	//Alarm
	TON_ComAlarm(IN:= MesWarningCom  , PT:= ParamTempoComAlarm, Q=>MesDataExd.MesAlarmCom) ;	// Alarms if ALL TRAM MODBUS did not work and timeout of 15s

// ALARM CODE //
	FB_AlarmCodeManager(
		bAlarm1			:= InvAlarm[1],		// All module are in alarm Inverter 1
		bAlarm2			:= InvAlarm[2],		// All module are in alarm Inverter 2
		bAlarm3			:= InvAlarm[3],		// All module are in alarm Inverter 3
		bAlarm4			:= MesDataExd.MesAlarmCom, 	//AT Least one Com error with 18 x Modules during more than 30s         
		bAlarm5			:= FALSE,
		bAlarm6			:= FALSE,
		bAlarm7			:= FALSE,
		bAlarm8			:= FALSE,
		bAlarm9			:= FALSE,
		bAlarm10		:= FALSE,
		bAlarm11		:= FALSE, 
		bAlarm12		:= FALSE, 
		bAlarm13		:= FALSE, 
		bAlarm14		:= FALSE, 													// 
		bAlarm15		:= FALSE,
		wAlarmCode		=> MesDataExd.MesAlarmCode);

// WARNING CODE //
	FB_AlarmCodeManager(
 		bAlarm1			:= INVWarning[1],//AT LEast one moduls of inverter 1 in alarm
		bAlarm2			:= INVWarning[2],//AT LEast one moduls of inverter 2 in alarm
		bAlarm3			:= INVWarning[3],//AT LEast one moduls of inverter 3 in alarm
		bAlarm4			:= MesWarningCom,//AT Least one Com error with 18 x Modules
		bAlarm5			:= FALSE, 		
		bAlarm6			:= FALSE, 		
		bAlarm7			:= FALSE, 
		bAlarm8			:= FALSE, 
		bAlarm9			:= FALSE, 
		bAlarm10		:= FALSE, 
		bAlarm11		:= FALSE, 
		bAlarm12		:= FALSE, 
		bAlarm13		:= FALSE, 
		bAlarm14		:= FALSE, 
		bAlarm15		:= FALSE, 
		wAlarmCode		=> MesDataExd.MesWarningCode);	

		
// EVENT CODE //
	FB_AlarmCodeManager(
		bAlarm1			:= RS_StartStop.Q1, 			// Start command
		bAlarm2			:= NOT RS_StartStop.Q1, 		// Stop command
		bAlarm3			:= FALSE,	
		bAlarm4			:= FALSE, 	
		bAlarm5			:= FALSE, 
		bAlarm6			:= FALSE, 
		bAlarm7			:= FALSE, 
		bAlarm8			:= FALSE, 
		bAlarm9			:= FALSE, 
		bAlarm10		:= FALSE, 
		bAlarm11		:= FALSE, 
		bAlarm12		:= FALSE, 
		bAlarm13		:= FALSE, 
		bAlarm14		:= FALSE, 
		bAlarm15		:= FALSE, 
		wAlarmCode		=> MesDataExd.MesEventCode);
END_METHOD

METHOD M_CP
//////////////////
//  Emulator
/////////////////

VAR 
	// Method local variables (reinitialized at each cycle) 
	
END_VAR


SUPER^.M_CP() ; 




Trig_Cmd_Read(CLK:=IN_CmdToggleRead);
//Trig_Cmd_Write(CLK:=IN_CmdToggleWrite);
//	
IF Trig_Cmd_Read.Q THEN
	IN_CmdToggleRead := FALSE;
	MesDataExd.AX_INV[1].MesData.MesCP_Read := NOT MesDataExd.AX_INV[1].MesData.MesCP_Read;
END_IF
//
//
//IF Trig_Cmd_Write.Q THEN
//	IN_CmdToggleWrite := FALSE;
//	MesDataExd.MesData.MesCP_Write := NOT MesDataExd.MesData.MesCP_Write;
//END_IF
END_METHOD

{attribute 'object_name' := 'M_Curtail'}
METHOD M_Curtail
//////////////////
// Write Curtail Command through modbus to PV inverters.  
//////////////////
VAR 
	// Method local variables (reinitialized at each cycle) 
	Threshold 			 : INT:=5 ;					// (0-100) Change percentage of Range to trigger the write command. 

	CHECK				 : BOOL; 					// Check if changes. 
	WriteCmdInvMode		: BOOL;

	MesSEPAM	: ProtectRelay_S48;
	

END_VAR




MesDataExd.OUT_SetptTanPhi := IN_SetptTanPhi ; 
MesDataExd.OUT_SetptP		:= ParamPn ; 
MesDataExd.OUT_CmdStart	:= TRUE ;
MesDataExd.OUT_CmdStop	:= FALSE ;

	
OUT_CmdSetpt420_IO := 32767- REAL_TO_INT((32767 * (MesDataExd.OUT_SetptTanPhi+0.484)/(0.968))  );		// ? ? 
 
SUPER^.M_Curtail() ;
END_METHOD

METHOD M_Execute
//////////////////
//  Method Calls 
/////////////////

VAR 
	// Method local variables (reinitialized at each cycle) 

END_VAR
IF  bInit THEN
	M_Init();
END_IF

(*
TP_Read(In := NOT(TP_Read.Q) AND NOT ReadBusy);
RTrig(CLK := TP_Read.Q);
ClockRead := RTrig.Q;
*)
SUPER^.M_Execute() ;
END_METHOD

METHOD M_Init
VAR_INPUT
END_VAR

VAR

END_VAR
//ParamPn := 990 ;
bInit := FALSE;
//FB_ModbusRTU() ;
AX_bRead[1] := TRUE ; 
(*
FB_ModbusRead(
	Inquantity		:= Nb_DataBlockModules,
	InUnitID 		:= ParamUnitID ,
	InTimeout		:= ParamTimeout,
	InInterfaceSub	:= FALSE,
	InFunctionRead	:= TRUE	);
	
	*)
END_METHOD

{attribute 'object_name' := 'M_Read'}
METHOD M_Read
//////////
// Read Method for SMA : Modbus reading
//////////
VAR
	// Method local variables (reinitialized at each cycle) 
	MW_32MLE		: FB_WordsToFloat32MLE;
	AX_bRead_init 		: ARRAY[0..18] OF BOOL; 
	KK					: BYTE;						 // Index to loop over modbus blocks. 	
	JJ					: BYTE;

	InclockRead: INT;
END_VAR


IF MesDataExd.AX_INV[1].MesData.MesCP_Read  THEN	







OutFBCompleteted:=FALSE;

// MODBUS REQUEST//


	
		// Reset Structure output. 
		//InputStructRead	:= InputStructRead_Null; 
		//
		//InputStructRead.InFunction := ParamFunctionReadModbus;
		//InputStructRead.InQuantity := Nb_DataBlockModules;	
		//
		//InputStructRead.OutBusy := ADR(ReadBusy);
		//InputStructRead.OutError := ADR(ReadError);
		//InputStructRead.OutCompleted := ADR(bReadCompleted);

		FB_ModbusRTU.ReadRTU1(
				InClockRead := NOT ClockRead AND AX_bRead[Steps],
				InStartAddr :=  AX_Start_Adresse[Steps],
				InQuantity := Nb_DataBlockModules,
				InUnitID := ParamUnitID,
				InTimeout := T#1500MS,
				InAddrDest := ADR(MesBlock_Temp[Steps]),
				InFunctionRead := ParamFunctionReadModbus,
				InInterfaceSub	:= FALSE 
			);
		
		IF  FB_ModbusRTU.ReadRTU1.OutBusy AND AX_bRead[Steps]THEN 
			AX_bRead[Steps] 	:= FALSE; 
		
		END_IF	
	
		RTrigI(CLK:= FB_ModbusRTU.ReadRTU1.TmpError );
		IF FB_ModbusRTU.ReadRTU1.OutbCompleted THEN

			Steps:= SEL(Steps >= 18 , Steps +1 , 1) ;
			AX_bRead[Steps] 	:= TRUE;
			ReadError := FALSE ; 
			
		ELSIF NOT FB_ModbusRTU.ReadRTU1.OutBusy  AND  RTrigI.Q THEN
			Steps:= SEL(Steps >= 18 , Steps +1 , 1) ;
			AX_bRead[Steps] 	:= TRUE;
			ReadError := TRUE ; 
		
		END_IF

//FB_ModbusRTU() ; 

	CalAllCompleted := AX_bRead[1] AND AX_bRead[2] AND AX_bRead[3] AND AX_bRead[4] AND AX_bRead[5] AND AX_bRead[6]; 
	CalAllCompleted := CalAllCompleted AND AX_bRead[7] AND AX_bRead[8] AND AX_bRead[9] AND AX_bRead[10] AND AX_bRead[11] AND AX_bRead[12];
	CalAllCompleted := CalAllCompleted AND AX_bRead[13] AND AX_bRead[14] AND AX_bRead[15] AND AX_bRead[16] AND AX_bRead[17] AND AX_bRead[18];	
	
	CalAllBugged	:= AX_bRead[1] OR AX_bRead[2] OR AX_bRead[3] OR AX_bRead[4] OR AX_bRead[5] OR AX_bRead[6];
	CalAllBugged 	:= CalAllBugged OR AX_bRead[7] OR AX_bRead[8] OR AX_bRead[9] OR AX_bRead[10] OR AX_bRead[11] OR AX_bRead[12];
	CalAllBugged 	:= CalAllBugged OR AX_bRead[13] OR AX_bRead[14] OR AX_bRead[15] OR AX_bRead[16] OR AX_bRead[17] OR AX_bRead[18];	
	
	
	OutFBCompleteted := CalAllCompleted	;
	TON_AllBugged(IN := NOT CalAllBugged, pt := T#10S);
	TRIG_AllBugged(CLK := TON_AllBugged.Q);
	IF TRIG_AllBugged.Q THEN
		TON_AllBugged(IN := FALSE);
		AX_bRead[Steps] := TRUE;
	END_IF

	////CHECK IF ALL MODBUS REQUESTS ARE FINISHED
	IF (CalAllCompleted) THEN
		////RESETING CLOCK READ FOR EACH REQUEST
		//AX_bRead:= AX_bRead_init;
		CalAllCompleted := FALSE;
	END_IF
	MesTempPos[1] := 0;
	MesTempPos[2] := 0;
	// PROPERTIES UPDATE
	// MODBUS BLOCKS SEPARATION	& PROPERTIES UPDATE
		//INVERTER 01 - Module
	
	
	JJ := 1 ; 
	
	FOR KK := 1 TO 18 BY 1 DO
		
		IF KK =1 THEN
			//InverterNumber := 1 ;
			InverterNumber := 1;// on constate un décalage de deux bloque avec cette méthode. Ainsi , l'adresse correspondant à INV1 (AX_Start_Adresse[1] , donne un résultat dans le block 3 Block_Temp[3]. 

		END_IF

		DecalageInvModule := SEL(((KK+0) MOD 6) =0 , (KK+0) MOD 6  , 6);//KK - (6*(InverterNumber-1)) ;
			
		//Word on 1 register To INT 
		MesDataExd.AX_INV[InverterNumber].AX_PowerCol[DecalageInvModule].MesSN 				:= WORD_TO_INT(MesBlock_Temp[KK][0]);
		MesDataExd.AX_INV[InverterNumber].AX_PowerCol[DecalageInvModule].MesID_Type 	:= WORD_TO_INT(MesBlock_Temp[KK][1]);
		MesDataExd.AX_INV[InverterNumber].AX_PowerCol[DecalageInvModule].MesID_StateGlobal		:= WORD_TO_INT(MesBlock_Temp[KK][2]);
		MesDataExd.AX_INV[InverterNumber].AX_PowerCol[DecalageInvModule].MesIDState	    := WORD_TO_INT(MesBlock_Temp[KK][3]);
		MesDataExd.AX_INV[InverterNumber].AX_PowerCol[DecalageInvModule].MesAlarmID		:= WORD_TO_INT(MesBlock_Temp[KK][4]);
		// 5 et 6 is blanck
		//Word on 2 register To Float 32
		//Module Information
			//Part1
		MW_32MLE(InFirstWord:=MesBlock_Temp[KK][7],InSecondWord:=MesBlock_Temp[KK][8],OutCalReal	=>MesDataExd.AX_INV[InverterNumber].AX_PowerCol[DecalageInvModule].MesEDay);
		MW_32MLE(InFirstWord:=MesBlock_Temp[KK][9],InSecondWord:=MesBlock_Temp[KK][10],OutCalReal	=>MesDataExd.AX_INV[InverterNumber].AX_PowerCol[DecalageInvModule].MesETot);
		MW_32MLE(InFirstWord:=MesBlock_Temp[KK][11],InSecondWord:=MesBlock_Temp[KK][12],OutCalReal  =>MesDataExd.AX_INV[InverterNumber].AX_PowerCol[DecalageInvModule].MesEPartial);
		MW_32MLE(InFirstWord:=MesBlock_Temp[KK][13],InSecondWord:=MesBlock_Temp[KK][14],OutCalReal  =>MesDataExd.AX_INV[InverterNumber].AX_PowerCol[DecalageInvModule].MesEWeek);
		MW_32MLE(InFirstWord:=MesBlock_Temp[KK][15],InSecondWord:=MesBlock_Temp[KK][16],OutCalReal  =>MesDataExd.AX_INV[InverterNumber].AX_PowerCol[DecalageInvModule].MesEMonth);
		MW_32MLE(InFirstWord:=MesBlock_Temp[KK][17],InSecondWord:=MesBlock_Temp[KK][18],OutCalReal  =>MesDataExd.AX_INV[InverterNumber].AX_PowerCol[DecalageInvModule].MesEYear);
			//Part2                                                                                                      
		MW_32MLE(InFirstWord:=MesBlock_Temp[KK][33],InSecondWord:=MesBlock_Temp[KK][34],OutCalReal  =>MesDataExd.AX_INV[InverterNumber].AX_PowerCol[DecalageInvModule].MesTemp_Inv);
		MW_32MLE(InFirstWord:=MesBlock_Temp[KK][35],InSecondWord:=MesBlock_Temp[KK][36],OutCalReal  =>MesDataExd.AX_INV[InverterNumber].AX_PowerCol[DecalageInvModule].MesTemp_Supply);
		MW_32MLE(InFirstWord:=MesBlock_Temp[KK][37],InSecondWord:=MesBlock_Temp[KK][38],OutCalReal  =>MesDataExd.AX_INV[InverterNumber].AX_PowerCol[DecalageInvModule].MesTemp_Headsink);
		MW_32MLE(InFirstWord:=MesBlock_Temp[KK][39],InSecondWord:=MesBlock_Temp[KK][40],OutCalReal  =>MesDataExd.AX_INV[InverterNumber].AX_PowerCol[DecalageInvModule].MesTemp_T2);
		MW_32MLE(InFirstWord:=MesBlock_Temp[KK][41],InSecondWord:=MesBlock_Temp[KK][42],OutCalReal  =>MesDataExd.AX_INV[InverterNumber].AX_PowerCol[DecalageInvModule].MesTemp_T3);
		

		// Detect Communication Error : MesID_StateGlobal = 0 , MesAlarmID = 0 , Temp_Inv = 0 
		IF MesDataExd.AX_INV[InverterNumber].AX_PowerCol[DecalageInvModule].MesTemp_Inv = 0 
			AND MesDataExd.AX_INV[InverterNumber].AX_PowerCol[DecalageInvModule].MesID_StateGlobal = 0 
			AND MesDataExd.AX_INV[InverterNumber].AX_PowerCol[DecalageInvModule].MesAlarmID = 0 THEN  
				MesDataExd.AX_INV[InverterNumber].AX_PowerCol[DecalageInvModule].MesAlarmID := 8 ; 
		END_IF
		
	
		IF  MesDataExd.AX_INV[InverterNumber].AX_PowerCol[DecalageInvModule].MesID_Type = 1  THEN
			//Slave
			MW_32MLE(InFirstWord:=MesBlock_Temp[KK][19],InSecondWord:=MesBlock_Temp[KK][20],OutCalReal=>MesDataExd.AX_INV[InverterNumber].AX_PowerCol[DecalageInvModule].MesV);
			MW_32MLE(InFirstWord:=MesBlock_Temp[KK][21],InSecondWord:=MesBlock_Temp[KK][22],OutCalReal=>MesTempPSlave[JJ][4]);
			MesDataExd.AX_INV[InverterNumber].AX_PowerCol[DecalageInvModule].MesI := MesTempPSlave[JJ][4] ; 
			MW_32MLE(InFirstWord:=MesBlock_Temp[KK][23],InSecondWord:=MesBlock_Temp[KK][24],OutCalReal=>MesTempPSlave[JJ][1]);
			MesDataExd.AX_INV[InverterNumber].AX_PowerCol[DecalageInvModule].MesData.MesP := MesTempPSlave[JJ][1];
			MW_32MLE(InFirstWord:=MesBlock_Temp[KK][25],InSecondWord:=MesBlock_Temp[KK][26],OutCalReal=>MesDataExd.AX_INV[InverterNumber].AX_PowerCol[DecalageInvModule].MesData.MesFreq);
			MW_32MLE(InFirstWord:=MesBlock_Temp[KK][27],InSecondWord:=MesBlock_Temp[KK][28],OutCalReal=>MesTempPSlave[JJ][2]);
			MesDataExd.AX_INV[InverterNumber].AX_PowerCol[DecalageInvModule].MesData.MesPdc := MesTempPSlave[JJ][2];
			MW_32MLE(InFirstWord:=MesBlock_Temp[KK][29],InSecondWord:=MesBlock_Temp[KK][30],OutCalReal=>MesDataExd.AX_INV[InverterNumber].AX_PowerCol[DecalageInvModule].MesData.MesUdc);
			MW_32MLE(InFirstWord:=MesBlock_Temp[KK][31],InSecondWord:=MesBlock_Temp[KK][32],OutCalReal=>MesTempPSlave[JJ][3]);
			MesDataExd.AX_INV[InverterNumber].AX_PowerCol[DecalageInvModule].MesData.MesIdc := MesTempPSlave[JJ][3] ;
		ELSE      
			//Master                                                                                                               
			MW_32MLE(InFirstWord:=MesBlock_Temp[KK][55],InSecondWord:=MesBlock_Temp[KK][56],OutCalReal=>MesDataExd.AX_INV[InverterNumber].AX_PowerCol[DecalageInvModule].MesV);
			MW_32MLE(InFirstWord:=MesBlock_Temp[KK][57],InSecondWord:=MesBlock_Temp[KK][58],OutCalReal=>MesTempPMaster[JJ][4]);
			MW_32MLE(InFirstWord:=MesBlock_Temp[KK][59],InSecondWord:=MesBlock_Temp[KK][60],OutCalReal=>MesTempPMaster[JJ][1]);
			//MesDataExd.AX_INV[InverterNumber].AX_PowerCol[DecalageInvModule].MesP := MesTempPMaster[JJ][1];
			MW_32MLE(InFirstWord:=MesBlock_Temp[KK][25],InSecondWord:=MesBlock_Temp[KK][26],OutCalReal=>MesDataExd.AX_INV[InverterNumber].AX_PowerCol[DecalageInvModule].MesData.MesFreq);
			MW_32MLE(InFirstWord:=MesBlock_Temp[KK][61],InSecondWord:=MesBlock_Temp[KK][62],OutCalReal=>MesTempPMaster[JJ][2]);
			//MesDataExd.AX_INV[InverterNumber].AX_PowerCol[DecalageInvModule].MesPdc := MesTempPMaster[JJ][2];
			MW_32MLE(InFirstWord:=MesBlock_Temp[KK][63],InSecondWord:=MesBlock_Temp[KK][64],OutCalReal=>MesDataExd.AX_INV[InverterNumber].AX_PowerCol[DecalageInvModule].MesData.MesUdc);
			MW_32MLE(InFirstWord:=MesBlock_Temp[KK][65],InSecondWord:=MesBlock_Temp[KK][66],OutCalReal=>MesTempPMaster[JJ][3]); 
			MesTempPos[JJ] := DecalageInvModule ; 	// Relative Number of master module 
		END_IF
		
		IF KK MOD 2 =0 THEN
			IF Master_slave_Calculation AND MesTempPos[JJ]>0 THEN
				MesDataExd.AX_INV[InverterNumber].AX_PowerCol[MesTempPos[JJ]].MesData.MesP := MesTempPMaster[JJ][1]- MesTempPSlave[JJ][1];	// P
				MesDataExd.AX_INV[InverterNumber].AX_PowerCol[MesTempPos[JJ]].MesData.MesPdc := MesTempPMaster[JJ][2]- MesTempPSlave[JJ][2];	// Pdc
				MesDataExd.AX_INV[InverterNumber].AX_PowerCol[MesTempPos[JJ]].MesData.MesIdc :=MesTempPMaster[JJ][3]- MesTempPSlave[JJ][3];	// Idc
				MesDataExd.AX_INV[InverterNumber].AX_PowerCol[MesTempPos[JJ]].MesI := MesTempPMaster[JJ][4]- MesTempPSlave[JJ][4];	// I

				IF MesDataExd.AX_INV[InverterNumber].AX_PowerCol[MesTempPos[JJ]].MesData.MesP < 0 THEN 
					MesDataExd.AX_INV[InverterNumber].AX_PowerCol[MesTempPos[JJ]].MesData.MesP := 0 ; 
					MesDataExd.AX_INV[InverterNumber].AX_PowerCol[MesTempPos[JJ]].MesData.MesPdc := 0 ; 
					MesDataExd.AX_INV[InverterNumber].AX_PowerCol[MesTempPos[JJ]].MesData.MesIdc := 0 ; 
					MesDataExd.AX_INV[InverterNumber].AX_PowerCol[MesTempPos[JJ]].MesI := 0 ;
					MesDataExd.AX_INV[InverterNumber].AX_PowerCol[MesTempPos[JJ]].MesAlarmID := 8  ;  // Com error with master
					
				ELSIF MesDataExd.AX_INV[InverterNumber].AX_PowerCol[MesTempPos[JJ]].MesData.MesP > 50 THEN // Higher than Pnom 
					MesDataExd.AX_INV[InverterNumber].AX_PowerCol[MesTempPos[JJ]].MesAlarmID := 88  ; // Com error with Slave device 
				END_IF
				
			ELSIF MesTempPos[JJ]>0 THEN 
				MesDataExd.AX_INV[InverterNumber].AX_PowerCol[MesTempPos[JJ]].MesData.MesP := MesTempPMaster[JJ][1];	// P
				MesDataExd.AX_INV[InverterNumber].AX_PowerCol[MesTempPos[JJ]].MesData.MesPdc := MesTempPMaster[JJ][2];	// Pdc
				MesDataExd.AX_INV[InverterNumber].AX_PowerCol[MesTempPos[JJ]].MesData.MesIdc := MesTempPMaster[JJ][3];	// Idc				
				MesDataExd.AX_INV[InverterNumber].AX_PowerCol[MesTempPos[JJ]].MesI := MesTempPMaster[JJ][4];	// I					
				
			END_IF
			JJ := JJ +1;		
		END_IF
		
		// RACK informations
		IF DecalageInvModule = 6  THEN
			
			MW_32MLE(InFirstWord:=MesBlock_Temp[KK][43],InSecondWord:=MesBlock_Temp[KK][44],OutCalReal=>MesDataExd.AX_INV[InverterNumber].MesEDay);
			MW_32MLE(InFirstWord:=MesBlock_Temp[KK][45],InSecondWord:=MesBlock_Temp[KK][46],OutCalReal=>MesDataExd.AX_INV[InverterNumber].MesETot);
			MW_32MLE(InFirstWord:=MesBlock_Temp[KK][47],InSecondWord:=MesBlock_Temp[KK][48],OutCalReal=>MesDataExd.AX_INV[InverterNumber].MesEPartial);
			MW_32MLE(InFirstWord:=MesBlock_Temp[KK][49],InSecondWord:=MesBlock_Temp[KK][50],OutCalReal=>MesDataExd.AX_INV[InverterNumber].MesEWeek);
			MW_32MLE(InFirstWord:=MesBlock_Temp[KK][51],InSecondWord:=MesBlock_Temp[KK][52],OutCalReal=>MesDataExd.AX_INV[InverterNumber].MesEMonth);
			MW_32MLE(InFirstWord:=MesBlock_Temp[KK][53],InSecondWord:=MesBlock_Temp[KK][54],OutCalReal=>MesDataExd.AX_INV[InverterNumber].MesEYear);
			InverterNumber := SEL(InverterNumber=3 , InverterNumber + 1,1);
		END_IF
		
	END_FOR;
	
	//Calculation of Master/slave power
(*
	IF FALSE AND Master_slave_Calculation THEN
		//Inverter 1
			//P
			MesDataExd.AX_INV[1].AX_PowerCol[MesTempPos[1]].MesP := MesTempPMaster[1][1]- MesTempPSlave[1][1];
			MesDataExd.AX_INV[1].AX_PowerCol[MesTempPos[2]].MesP := MesTempPMaster[2][1]- MesTempPSlave[2][1];
			MesDataExd.AX_INV[1].AX_PowerCol[MesTempPos[3]].MesP := MesTempPMaster[3][1]- MesTempPSlave[3][1];
			//Pdc
			MesDataExd.AX_INV[1].AX_PowerCol[MesTempPos[1]].MesPdc := MesTempPMaster[1][2]- MesTempPSlave[1][2];
			MesDataExd.AX_INV[1].AX_PowerCol[MesTempPos[2]].MesPdc := MesTempPMaster[2][2]- MesTempPSlave[2][2];
			MesDataExd.AX_INV[1].AX_PowerCol[MesTempPos[3]].MesPdc := MesTempPMaster[3][2]- MesTempPSlave[3][2];
			
		//Inverter 2
			//P
			MesDataExd.AX_INV[2].AX_PowerCol[MesTempPos[4]].MesP := MesTempPMaster[4][1]- MesTempPSlave[4][1];
			MesDataExd.AX_INV[2].AX_PowerCol[MesTempPos[5]].MesP := MesTempPMaster[5][1]- MesTempPSlave[5][1];
			MesDataExd.AX_INV[2].AX_PowerCol[MesTempPos[6]].MesP := MesTempPMaster[6][1]- MesTempPSlave[6][1];
			//Pdc    
			MesDataExd.AX_INV[2].AX_PowerCol[MesTempPos[4]].MesPdc := MesTempPMaster[4][2]- MesTempPSlave[4][2];
			MesDataExd.AX_INV[2].AX_PowerCol[MesTempPos[5]].MesPdc := MesTempPMaster[5][2]- MesTempPSlave[5][2];
			MesDataExd.AX_INV[2].AX_PowerCol[MesTempPos[6]].MesPdc := MesTempPMaster[6][2]- MesTempPSlave[6][2];
		             
		//Inverter 3  
			//P       
			MesDataExd.AX_INV[3].AX_PowerCol[MesTempPos[7]].MesP := MesTempPMaster[7][1]- MesTempPSlave[7][1];
			MesDataExd.AX_INV[3].AX_PowerCol[MesTempPos[8]].MesP := MesTempPMaster[8][1]- MesTempPSlave[8][1];
			MesDataExd.AX_INV[3].AX_PowerCol[MesTempPos[9]].MesP := MesTempPMaster[9][1]- MesTempPSlave[9][1];
			//Pdc     
			MesDataExd.AX_INV[3].AX_PowerCol[MesTempPos[7]].MesPdc := MesTempPMaster[7][2]- MesTempPSlave[7][2];
			MesDataExd.AX_INV[3].AX_PowerCol[MesTempPos[8]].MesPdc := MesTempPMaster[8][2]- MesTempPSlave[8][2];
			MesDataExd.AX_INV[3].AX_PowerCol[MesTempPos[9]].MesPdc := MesTempPMaster[9][2]- MesTempPSlave[9][2];
	ELSE
		//Inverter 1
			MesDataExd.AX_INV[1].AX_PowerCol[MesTempPos[1]].MesP := MesTempPMaster[1][1];
			MesDataExd.AX_INV[1].AX_PowerCol[MesTempPos[2]].MesP := MesTempPMaster[2][1];
			MesDataExd.AX_INV[1].AX_PowerCol[MesTempPos[3]].MesP := MesTempPMaster[3][1];
			//Pdc     
			MesDataExd.AX_INV[1].AX_PowerCol[MesTempPos[1]].MesPdc := MesTempPMaster[1][2];
			MesDataExd.AX_INV[1].AX_PowerCol[MesTempPos[2]].MesPdc := MesTempPMaster[2][2];
			MesDataExd.AX_INV[1].AX_PowerCol[MesTempPos[3]].MesPdc := MesTempPMaster[3][2];
		//Inverter 2  
			//P      
			MesDataExd.AX_INV[2].AX_PowerCol[MesTempPos[4]].MesP := MesTempPMaster[4][1];
			MesDataExd.AX_INV[2].AX_PowerCol[MesTempPos[5]].MesP := MesTempPMaster[5][1];
			MesDataExd.AX_INV[2].AX_PowerCol[MesTempPos[6]].MesP := MesTempPMaster[6][1];
			//Pdc     
			MesDataExd.AX_INV[2].AX_PowerCol[MesTempPos[4]].MesPdc := MesTempPMaster[4][2];
			MesDataExd.AX_INV[2].AX_PowerCol[MesTempPos[5]].MesPdc := MesTempPMaster[5][2];
			MesDataExd.AX_INV[2].AX_PowerCol[MesTempPos[6]].MesPdc := MesTempPMaster[6][2];
		             
		//Inverter 3  
			//P      
			MesDataExd.AX_INV[3].AX_PowerCol[MesTempPos[7]].MesP := MesTempPMaster[7][1];
			MesDataExd.AX_INV[3].AX_PowerCol[MesTempPos[8]].MesP := MesTempPMaster[8][1];
			MesDataExd.AX_INV[3].AX_PowerCol[MesTempPos[9]].MesP := MesTempPMaster[9][1];
			//Pdc     
			MesDataExd.AX_INV[3].AX_PowerCol[MesTempPos[7]].MesPdc := MesTempPMaster[7][2];
			MesDataExd.AX_INV[3].AX_PowerCol[MesTempPos[8]].MesPdc := MesTempPMaster[8][2];
			MesDataExd.AX_INV[3].AX_PowerCol[MesTempPos[9]].MesPdc := MesTempPMaster[9][2];
	END_IF	
	*)
//Addition des puissance
	FOR KK:= 1 TO 3 DO 
		MesDataExd.AX_INV[KK].MesData.MesP := 0 ; 
		MesDataExd.AX_INV[KK].MesData.MesI := 0 ; 
		MesDataExd.AX_INV[KK].MesData.MesPdc := 0 ; 
		MesDataExd.AX_INV[KK].MesData.MesFreq :=  0 ; 
		MesDataExd.AX_INV[KK].MesData.MesIdc := 0  ; 
		MesDataExd.AX_INV[KK].MesData.MesV := 0  ; 		
		MesDataExd.AX_INV[KK].MesData.MesUdc := 0  ; 		
 		MesDataExd.AX_INV[KK].MesData.MesTemp	:= 0 ; 
		MesDataExd.AX_INV[KK].MesData.ParamPn := ParamPn/3 ; 
		
		FOR InclockRead:= 1 TO 6 DO 
			MesDataExd.AX_INV[KK].MesData.MesP  	:= MesDataExd.AX_INV[KK].MesData.MesP +	MesDataExd.AX_INV[KK].AX_PowerCol[InclockRead].MesData.MesP ;					
			MesDataExd.AX_INV[KK].MesData.MesPdc  	:= MesDataExd.AX_INV[KK].MesData.MesPdc +	MesDataExd.AX_INV[KK].AX_PowerCol[InclockRead].MesData.MesPdc ;					
			MesDataExd.AX_INV[KK].MesData.MesI  	:= MesDataExd.AX_INV[KK].MesData.MesI +	MesDataExd.AX_INV[KK].AX_PowerCol[InclockRead].MesI ;					
			MesDataExd.AX_INV[KK].MesData.MesFreq 	:= MAX(MesDataExd.AX_INV[KK].MesData.MesFreq , MesDataExd.AX_INV[KK].AX_PowerCol[InclockRead].MesData.MesFreq) ; 
			MesDataExd.AX_INV[KK].MesData.MesIdc  	:= MesDataExd.AX_INV[KK].MesData.MesIdc +	MesDataExd.AX_INV[KK].AX_PowerCol[InclockRead].MesData.MesIdc ;			
			MesDataExd.AX_INV[KK].MesData.MesUdc 	:= MAX(MesDataExd.AX_INV[KK].MesData.MesUdc , MesDataExd.AX_INV[KK].AX_PowerCol[InclockRead].MesData.MesUdc) ; 		
			MesDataExd.AX_INV[KK].MesData.MesV 	:= MAX(MesDataExd.AX_INV[KK].MesData.MesV , MesDataExd.AX_INV[KK].AX_PowerCol[InclockRead].MesV) ; 
			MesDataExd.AX_INV[KK].MesData.MesTemp 	:= MAX(MesDataExd.AX_INV[KK].MesData.MesTemp , MesDataExd.AX_INV[KK].AX_PowerCol[InclockRead].MesTemp_Inv) ; 	
		END_FOR
	

	END_FOR

END_IF
END_METHOD

METHOD M_StateManager
//////////////////
// Detect which is the state of the inverter. IF loss of communication MesState =0 , the last inverter state is kept .  
/////////////////

VAR 
	// Method local variables (reinitialized at each cycle) 

	
	KK: INT;
	LL: INT;

	MesAll_Start	: BOOL;
	MesALO_Fault 	: BOOL;
	MesALO_Stopped	: BOOL;
	MesAll_Fault: BOOL;
	
	
	CalIDState_PowerCol: INT;
	CalNbPowerCol: INT;	
	
	
END_VAR
MesDataExd.MesNbInvConnected := 0  ; 
FOR KK:= 1  TO 3 DO 
	MesDataExd.AX_INV[KK].MesNbPowerColConnected := 0  ; 
	FOR LL:=1 TO 6 DO 
		
		CalIDState_PowerCol := MesDataExd.AX_INV[KK].AX_PowerCol[LL].MesID_StateGlobal ; 
	
		IF CalIDState_PowerCol = 6 THEN 
			MesDataExd.AX_INV[KK].MesNbPowerColConnected  := MesDataExd.AX_INV[KK].MesNbPowerColConnected + 1 ; 
		END_IF

	END_FOR	
	
	IF MesDataExd.AX_INV[KK].MesNbPowerColConnected> 0  THEN 
		MesDataExd.MesNbInvConnected := MesDataExd.MesNbInvConnected  + 1 ;  
	END_IF

END_FOR

// Check over all the powercolonnes 
//O=Stopped, 1 = MPPT, 2 = Sleeping, 3 = Starting, 4 = Throttled, 5 = Shutting down, 6 = Fault, 7 = Standby

FOR KK := 1 TO CstNbInv_PTR_G DO
	MesAll_Start := TRUE;
	MesAll_Fault := TRUE ;
	FOR LL := 1 TO CstNbPowerCol_INV_G DO 
		MesAll_Start := MesAll_Start AND MesDataExd.AX_INV[KK].AX_PowerCol[LL].MesIDState = 45;
		MesALO_Fault := MesALO_Fault OR MesDataExd.AX_INV[KK].AX_PowerCol[LL].MesAlarmID > 0;
		MesAll_Fault := MesAll_Fault AND MesDataExd.AX_INV[KK].AX_PowerCol[LL].MesAlarmID > 0;
		MesALO_Stopped := MesALO_Stopped OR 
			(MesDataExd.AX_INV[KK].AX_PowerCol[LL].MesIDState = 45 AND MesDataExd.AX_INV[KK].AX_PowerCol[LL].MesAlarmID > 0);
	END_FOR
	
	MesDataExd.AX_INV[KK].MesData.MesState := 0;
	
	IF MesDataExd.AX_INV[KK].MesNbPowerColConnected > 0 THEN 
		IF MesDataExd.AX_INV[KK].MesData.MesP > 0.01 THEN 
			MesDataExd.AX_INV[KK].MesData.MesState.1 := TRUE ; // MPPT 
		ELSE 
			MesDataExd.AX_INV[KK].MesData.MesState.7 := TRUE ;  // Standby 
		END_IF 	
	ELSE 
		IF MesAll_Fault THEN 
			MesDataExd.AX_INV[KK].MesData.MesState.6 := TRUE ; // Fault 
		ELSE 
			MesDataExd.AX_INV[KK].MesData.MesState.0 := TRUE ; // Off 
		END_IF
	END_IF

END_FOR

MesDataExd.MesState 			:= 0  ; // At Cluster level
IF MesDataExd.MesNbInvConnected=0   THEN  // 
	// OFF State  
	MesDataExd.MesState.0 		:= 1 ; 
	
ELSE
	// ON State
	MesDataExd.MesState.2 		:= 1 ;
	
END_IF



SUPER^.M_StateManager() ;
END_METHOD

END_FUNCTION_BLOCK

// ---- 00_FunctionsBlocks/Beckhoff/Communication/ModbusRTU/FB_ModbusRTU.TcPOU
FUNCTION_BLOCK FB_ModbusRTU
// Send Modbus Read Request for the first element of the buffer . Then remove the first line when executed ( busy)  and move all the other line to the left. Position 2 becomes position 1 , ...
VAR CONSTANT
	NbElementsBuffer				: UINT := 20;
	
END_VAR
VAR_INPUT PERSISTENT
	ParamTimeout					: TIME := T#500MS;
	ParamInterfaceSub				: BOOL;
END_VAR
VAR
	Buffer 							: ARRAY[1..NbElementsBuffer] OF Struct_InputRTU ; // Buffer to store actions
	Priority 						: ARRAY[1..NbElementsBuffer] OF UINT; // Array to store priorities
	InitialStruct 					: Struct_InputRTU;
	bInit 							: BOOL;
	ReadRTU1						: FB_ReadModbusRTU_V2;

	KK : UINT;
	
	pBoolNull						: BOOL;
	pIntNull						: INT;
	pArrayNull						: BYTE;

	R_TRIG_Error					: R_TRIG ;
	F_Trig_busy						: F_TRIG;
END_VAR

IF NOT bInit THEN
	// Empty all structures . 
	M_Init();
ELSE
	
		// ATTENTION , IL NE FAUT PAS ENVOYER UN NOUVEAU MODBUS TANT QUE LE PRECEDENT N EST PAS FINI DE TRAITER .DE MEME IL NE FAUT PAS QUE LE CYCLE D AJOUT DU FIFO SOIT PLUS RAPIDE QUE LE TRAITEMENT DU RTU 
		// TEmpo de 30 s apres une alarmes avant de refaire un essai . il ne faudrait pas que ca bloque les autres commandes .  

		IF priority[1] <> 0 THEN

			ReadRTU1(
				InClockRead := TRUE,
				InStartAddr := Buffer[1].InStartAddr,
				InQuantity := Buffer[1].InQuantity,
				InUnitID := Buffer[1].InUnitID,
				InTimeout := ParamTimeout,
				InAddrDest := Buffer[1].InBuffer,
				InFunctionRead := Buffer[1].InFunction,
				InInterfaceSub	:= ParamInterfaceSub 
			);
		END_IF
		
		
		
		MEMCPY(destAddr := Buffer[1].OutBusy, srcAddr := ADR(ReadRTU1.OutBusy), n := SIZEOF(ReadRTU1.OutBusy));		

		//R_TRIG_Error(CLK:= ReadRTU1.OutErrorMbRead) ; 
		F_Trig_busy(clk := ReadRTU1.OutBusy);
		IF F_Trig_busy.Q THEN	// La lecture s 'est terminée par une erreur ou correcteemnt, on passe à l'element du buffer suivant . 
			MEMCPY(destAddr := Buffer[1].OutError, srcAddr := ADR(ReadRTU1.OutErrorMbRead), n := SIZEOF(ReadRTU1.OutErrorMbRead)); // Copy the errOR  
			MEMCPY(destAddr := Buffer[1].OutErrorId, srcAddr := ADR(ReadRTU1.OutErrorId), n := SIZEOF(ReadRTU1.OutErrorId));
			MEMCPY(destAddr := Buffer[1].OutCompleted, srcAddr := ADR(ReadRTU1.OutbCompleted), n := SIZEOF(ReadRTU1.OutbCompleted));	
			ReadRTU1.InClockRead := FALSE ; 
			ReadRTU1.Reset		:= TRUE ; 
			M_DeleteAction(InLigne := 1);
			//R_TRIG_Error(CLK:= FALSE ) ; 
			
		END_IF
END_IF

METHOD M_AddAction_FIFO : UINT //Method to add an element with a priority using FIFO strategy

VAR_INPUT
	InStruct 		: Struct_InputRTU;		// Structure input
	InPriority 		: UINT;					// Strategy input
END_VAR
VAR_OUTPUT
	OutBusy 		: BOOL;					// Output state of the Method
	OutError 		: BOOL;					// Output error of the Method
	OutErrorID 		: UINT;					//1: Empty input 2: Full Buffer
	OutCompleted 	: BOOL;					// Output state of the Method : not busy and no error
END_VAR
VAR
	KK 				: UINT;
	LineToDelete	: UINT;
END_VAR
OutError 	:= FALSE;
OutBusy 	:= TRUE;

IF NOT (CheckStruct(InStruct1 := InitialStruct, InStruct2 := InStruct)) AND InPriority <> 0 THEN 			// Check that we don't input an empty value
	IF CheckStruct(InStruct1 := buffer[NbElementsBuffer], InStruct2 := InitialStruct) THEN 			// Check that the buffer isn't already full
		FOR KK := 1 TO NbElementsBuffer - 1 DO
			IF NOT CheckStruct(InStruct1 := buffer[NbElementsBuffer-KK], InStruct2 := InitialStruct) AND Priority[NbElementsBuffer-KK] > InPriority THEN 			// If the next position isn't empty  
				buffer[NbElementsBuffer-KK+1] := buffer[NbElementsBuffer-KK]; 		// I replace this position by the next  ( CE PREMIER IF N EST PAS EXECUTER SI TOUTES LES PRIORITES SONT IDENTIQUES . )
				Priority[NbElementsBuffer -KK +1 ] := Priority[NbElementsBuffer-KK];
			ELSE
				IF NOT CheckStruct(InStruct1 := buffer[NbElementsBuffer-KK], InStruct2 := InitialStruct) THEN		// Detect for buffer element that is not empty and assign new element to read to it. 
					buffer[NbElementsBuffer-KK+1] 	:= InStruct;
					M_AddAction_FIFO 				:= NbElementsBuffer-KK+1;
					Priority[NbElementsBuffer-KK+1] := InPriority;
					OutCompleted 		:= TRUE;
					EXIT ;
				END_IF
			END_IF
		END_FOR
		IF NOT Outcompleted THEN
			buffer[1] := InStruct;
			Priority[1] := InPriority;
			OutCompleted := TRUE;
			M_AddAction_Fifo := 1;
		END_IF
	ELSE
		OutErrorID 	:= 2;
		OutError 	:= TRUE;
	END_IF
ELSE
	OutErrorID 	:= 1;
	OutError 	:= TRUE;
END_IF
IF M_VerifActions(OutLigne=>LineToDelete) THEN	// Verifie si il  n ya pas deux fois la meme ligne , sinon, supprime les lignes en doubles . En pratique, forcement la derniere ligne . 
	M_DeleteAction(InLigne := LineToDelete);
END_IF
OutBusy := FALSE;
END_METHOD

METHOD M_DeleteAction : BOOL
VAR_INPUT
	InLigne 	: UINT;			// Input Ligne to delete
END_VAR
VAR_OUTPUT
	OutBusy 		: BOOL;					// Output state of the Method
	OutError 		: BOOL;					// Output error of the Method
	OutErrorID 		: UINT;					// 1: InLigne greater than Buffer size, 2: The buffer ligne is already empty, 3: The buffer is full
	OutCompleted 	: BOOL;					// Output state of the Method : not busy and no error
	
END_VAR

VAR
	KK 				: UINT;
END_VAR
IF InLigne <= NbElementsBuffer THEN // Check the InLigne is in the range of the buffer
	IF NOT checkstruct(InStruct1 := buffer[InLigne], InStruct2 := InitialStruct) THEN	// Check that the buffer ligne is not already empty
		IF checkstruct(InStruct1 := buffer[NbElementsBuffer], InStruct2 := InitialStruct)THEN //check that the buffer is not full
			FOR KK := InLigne TO NbElementsBuffer -1 DO
				Buffer[KK] := buffer[KK + 1] ;
				Priority[KK] := Priority[KK + 1] ;
			END_FOR
		ELSE
			OutError := TRUE;
			OutBusy := FALSE;
			OutCompleted := FALSE;
			OutErrorID := 3;
		END_IF
	ELSE
		OutError := TRUE;
		OutCompleted := FALSE;
		OutBusy := TRUE;
		OutErrorID := 2;
		
	END_IF
ELSE
	OutCompleted := FALSE;
	OutError := TRUE;
	OutBusy := FALSE;
	OutErrorID := 1;
END_IF
END_METHOD

METHOD M_Init : BOOL
VAR
	InStruct : Struct_InputRTU;
END_VAR

// Initialize the structure with empty elements. 

InitialStruct.InBuffer := ADR(pArrayNull);
InitialStruct.OutBusy := ADR(pBoolNull);
InitialStruct.OutCompleted := ADR(pBoolNull);
InitialStruct.OutError := ADR(pBoolNull);
InitialStruct.OutErrorId := ADR(pIntNull);
FOR KK := 1 TO NbElementsBuffer DO 
	Buffer[KK] := InitialStruct;
END_FOR	

bInit := TRUE;
END_METHOD

METHOD M_VerifActions : BOOL // Verifies there is not repeat in the liste : TRUE = At least 2 elements are the same
VAR_OUTPUT
	OutLigne 	 : UINT;
END_VAR

VAR
	KK: UINT;
	JJ: UINT;
	CheckStructValue : BOOL;
END_VAR
FOR KK := 1 TO NbElementsBuffer DO
	FOR JJ := 1 + KK TO NbElementsBuffer DO
		IF CheckStruct(InStruct1 := InitialStruct, instruct2 := buffer[KK]) THEN
			EXIT;
		ELSE
			CheckStructValue :=  checkstruct(InStruct1 := buffer[JJ], InStruct2 := buffer[KK]);
			M_VerifActions := M_VerifActions OR (CheckStructValue ) ;
			OutLigne := SEL(CheckStructValue AND Priority[KK]> priority[JJ], KK, JJ);
		END_IF
	END_FOR
END_FOR
END_METHOD

END_FUNCTION_BLOCK

// ---- 00_FunctionsBlocks/Beckhoff/Communication/ModbusRTU/FB_ReadModbusRTU_V2.TcPOU
FUNCTION_BLOCK FB_ReadModbusRTU_V2
/////////////////////////////////////////////////////////////////////// 
///////Read Modbus RTU on Rising Edge of Trigger ClockRead ////////
//If there is lost of communication, ParamNbAlms then if still 
//error wait ParamTimeRetry then loop 
//Version : V1.1
///////////////////////////////////////////////////////////////////////

VAR_INPUT
	InClockRead 			: BOOL;  		// Boolean to start the read
	InStartAddr				: WORD;  		// First address of the block
	InQuantity			    : WORD;	 		// Quantity of registers to read
	InUnitID				: BYTE ; 		// Unit Id of the Slave to be read
	InTimeout 				: TIME:=T#2S;   // Timeout param for the read
	InAddrDest		        : POINTER TO BYTE;
	InInterfaceSub			: BOOL:=FALSE;   // Serial interface RS422/RS485 TYPE (0:EL6021,1:SUB9)
	InFunctionRead          : UINT;          // 0 := ReadInputRegs, 1 := ReadRegs 
	ParamEnableRetryPause	: BOOL ; 
	Reset					: BOOL ;
END_VAR

VAR_OUTPUT
	OutErrorMbRead  		: BOOL; 	                // Alarm if three modbus attempts failed.
	OutBusy					: BOOL;					    //Busy
	OutErrorId				: INT;            //Id number of the error based on TC
	OutbCompleted			: BOOL;
	TmpError				: BOOL;	
END_VAR

VAR
	//Parameters
	ParamNbAlms				: UINT := 3;				// Parameter for the number of retries before the alarme
	ParamTimeRetry 			: TIME:=T#30S;				//Time to wait before a retry
	
	//Instantiation of FB
	MB 						: ModbusRtuMaster_PcCOM; 		// Multiple registers reading FROM SUB9 Interface
	MB_EL					: ModbusRtuMasterV2_KL6x22B;  // Multiple registers reading FROM EL6021 Interface
	R_TRIG          		: R_TRIG; 					// Rising edge detection for the trigger.
	TempoRetry      		: TP;
	
	//Variables of the code 
	Step            		: INT; 		    			// Grafcet step
	AlarmCounter    		: UINT; 					// Alarm Counter. Incremennted if modbus errOR  Alarm if counter =3 , resetable.  
	bRetry          		: BOOL:= FALSE; 			// Boolean to denote the retries
	
	TmpBusy					: BOOL;
	TmpErrorId				: INT;	
	
	TON_ReadRTU						: TON; 
END_VAR

OutbCompleted:= FALSE;
// RESET //
	IF Reset THEN 
			AlarmCounter		:= MAX(0,AlarmCounter-1) ;	// on enleve 1 au compteur pour supprimer l'alamrme. 
			OutErrorId 			:= 0 ; 
			OutErrorMbRead 	:=FALSE;
			Reset 				:= FALSE;
	END_IF
	
// ALARM MANAGEMENT //
TempoRetry(PT := ParamTimeRetry);
IF AlarmCounter = ParamNbAlms THEN 
	OutErrorMbRead 	:=TRUE;
	bRetry := SEL(ParamEnableRetryPause , FALSE ,  TRUE);		// False = disable retry 	
ELSE
	bRetry := FALSE;
	
END_IF

	// MODBUS SEQUENCE //
	
	IF InInterfaceSub THEN 

		CASE step OF
			0://Idle
				R_TRIG(CLK := InClockRead);
				IF R_TRIG.Q THEN 
					R_TRIG(CLK := FALSE);
					Step :=1;
					OutBusy         := TRUE;
				END_IF
			1 ://Processing Reply  
				TON_ReadRTU(IN:= TRUE , PT:= InTimeout + T#100MS ) ; // Overlay timeout . 
				CASE InFunctionRead OF
					1: 
						MB.ReadCoils
						(
							UnitID := InUnitId, 
							Quantity := InQuantity, 
							MBAddr := InStartAddr, 
							cbLength := 2* InQuantity, 
							pMemoryAddr := InAddrDest, 
							Execute := TRUE, 
							Timeout := InTimeout,
							Error => TmpError,
							Busy => TmpBusy,
							ErrorId => TmpErrorId,
						);	
					2:
						MB.ReadInputStatus
						(
							UnitID := InUnitId, 
							Quantity := InQuantity, 
							MBAddr := InStartAddr, 
							cbLength := 2* InQuantity, 
							pMemoryAddr := InAddrDest, 
							Execute := TRUE, 
							Timeout := InTimeout,
							Error => TmpError,
							Busy => TmpBusy,
							ErrorId => TmpErrorId,
						);	
					3:
						MB.ReadRegs
						(
							UnitID := InUnitId, 
							Quantity := InQuantity, 
							MBAddr := InStartAddr, 
							cbLength := 2* InQuantity, 
							pMemoryAddr := InAddrDest, 
							Execute := TRUE, 
							Timeout := InTimeout,
							Error => TmpError,
							Busy => TmpBusy,
							ErrorId => TmpErrorId,
						  );
					4:
						MB.ReadInputRegs
						(
							UnitID := InUnitId, 
							Quantity := InQuantity, 
							MBAddr := InStartAddr, 
							cbLength := 2* InQuantity, 
							pMemoryAddr := InAddrDest, 
							Execute := TRUE, 
							Timeout := InTimeout,
							Error => TmpError,
							Busy => TmpBusy,
							ErrorId => TmpErrorId,
						);
					5:
						MB.WriteSingleCoil
						(
							UnitID := InUnitId, 
							Quantity := InQuantity, 
							MBAddr := InStartAddr, 
							cbLength := 2* InQuantity, 
							pMemoryAddr := InAddrDest, 
							Execute := TRUE, 
							Timeout := InTimeout,
							Error => TmpError,
							Busy => TmpBusy,
							ErrorId => TmpErrorId,
						);
					6:
						MB.WriteSingleRegister
						(
							UnitID := InUnitId, 
							Quantity := InQuantity, 
							MBAddr := InStartAddr, 
							cbLength := 2* InQuantity, 
							pMemoryAddr := InAddrDest, 
							Execute := TRUE, 
							Timeout := InTimeout,
							Error => TmpError,
							Busy => TmpBusy,
							ErrorId => TmpErrorId,
						);
					15:
						MB.WriteMultipleCoils
						(
							UnitID := InUnitId, 
							Quantity := InQuantity, 
							MBAddr := InStartAddr, 
							cbLength := 2* InQuantity, 
							pMemoryAddr := InAddrDest, 
							Execute := TRUE, 
							Timeout := InTimeout,
							Error => TmpError,
							Busy => TmpBusy,
							ErrorId => TmpErrorId,
						);
					16:
						MB.WriteRegs
						(
							UnitID := InUnitId, 
							Quantity := InQuantity, 
							MBAddr := InStartAddr, 
							cbLength := 2* InQuantity, 
							pMemoryAddr := InAddrDest, 
							Execute := TRUE, 
							Timeout := InTimeout,
							Error => TmpError,
							Busy => TmpBusy,
							ErrorId => TmpErrorId,
						);
				END_CASE
				
				IF NOT (TmpBusy) AND NOT (TmpError) THEN
					TempoRetry(In:= FALSE);
					TON_ReadRTU(IN:= FALSE ) ; 
					MB.ReadInputRegs(Execute:= FALSE);
					MB.ReadRegs(Execute:= FALSE);
					MB.ReadCoils(Execute:= FALSE);
					MB.ReadInputStatus(Execute:= FALSE);
					MB.WriteSingleCoil(Execute:= FALSE);
					MB.WriteSingleRegister(Execute:= FALSE);
					MB.WriteMultipleCoils(Execute:= FALSE);
					MB.WriteRegs(Execute:= FALSE);
					OutErrorId 		:= 0;
					OutErrorMbRead	:= FALSE;
					AlarmCounter	:= 0; // Reset counter after successful modbus read. 
					OutbCompleted 	:= TRUE ; 
					Step 			:= 0;
					OutBusy         := FALSE;
				ELSIF ((NOT (TmpBusy) AND TmpError) OR TON_ReadRTU.Q)  AND NOT(bRetry) THEN
	
					TempoRetry(In:= FALSE);
					bRetry := FALSE;
					MB.ReadCoils(Execute:= FALSE);
					MB.ReadInputRegs(Execute:= FALSE);
					MB.ReadInputStatus(Execute:= FALSE);
					MB.ReadRegs(Execute:= FALSE);
					MB.WriteSingleCoil(Execute:= FALSE);
					MB.WriteSingleRegister(Execute:= FALSE);
					MB.WriteMultipleCoils(Execute:= FALSE);
					MB.WriteRegs(Execute:= FALSE);
					AlarmCounter 	:= MIN(AlarmCounter + 1,3) ; 
					OutErrorId		:= SEL(TON_ReadRTU.Q , TmpErrorId ,250 );
					Step 			:= 0;
					TON_ReadRTU(IN:= FALSE ) ; 
					OutBusy         := FALSE;
				ELSIF NOT (TmpBusy) AND TmpError AND bRetry THEN
					MB.ReadInputRegs(Execute:= FALSE);
					MB.ReadRegs(Execute:= FALSE);
					MB.ReadCoils(Execute:= FALSE);
					MB.ReadInputStatus(Execute:= FALSE);
					MB.WriteSingleCoil(Execute:= FALSE);
					MB.WriteSingleRegister(Execute:= FALSE);
					MB.WriteMultipleCoils(Execute:= FALSE);
					MB.WriteRegs(Execute:= FALSE);
					step := 2;
					OutBusy         := FALSE;
				END_IF	
			2: 
				TempoRetry(In:= TRUE);		// LEAVE SOME TIME BEFORE NEW ATTEMPT . 
				IF NOT(TempoRetry.Q) THEN
					TempoRetry(In:= FALSE);
					//AlarmCounter := 0;
					step := 0;
					
				END_IF
				
		END_CASE
	
	ELSE 
		
			CASE step OF
			0://Idle
				R_TRIG(CLK := InClockRead);
				IF R_TRIG.Q THEN 
					R_TRIG(CLK := FALSE);
					Step :=1;
					OutBusy         := TRUE;
				END_IF
			1 ://Processing Reply  
				TON_ReadRTU(IN:= TRUE , PT:= InTimeout + T#100MS ) ; // Overlay timeout . 
				CASE InFunctionRead OF
					1: 
						MB_EL.ReadCoils
						(
							UnitID := InUnitId, 
							Quantity := InQuantity, 
							MBAddr := InStartAddr, 
							cbLength := 2* InQuantity, 
							pMemoryAddr := InAddrDest, 
							Execute := TRUE, 
							Timeout := InTimeout,
							Error => TmpError,
							Busy => TmpBusy,
							ErrorId => TmpErrorId,
						);	
					2:
						MB_EL.ReadInputStatus
						(
							UnitID := InUnitId, 
							Quantity := InQuantity, 
							MBAddr := InStartAddr, 
							cbLength := 2* InQuantity, 
							pMemoryAddr := InAddrDest, 
							Execute := TRUE, 
							Timeout := InTimeout,
							Error => TmpError,
							Busy => TmpBusy,
							ErrorId => TmpErrorId,
						);	
					3:
						MB_EL.ReadRegs
						(
							UnitID := InUnitId, 
							Quantity := InQuantity, 
							MBAddr := InStartAddr, 
							cbLength := 2* InQuantity, 
							pMemoryAddr := InAddrDest, 
							Execute := TRUE, 
							Timeout := InTimeout,
							Error => TmpError,
							Busy => TmpBusy,
							ErrorId => TmpErrorId,
						  );
					4:
						MB_EL.ReadInputRegs
						(
							UnitID := InUnitId, 
							Quantity := InQuantity, 
							MBAddr := InStartAddr, 
							cbLength := 2* InQuantity, 
							pMemoryAddr := InAddrDest, 
							Execute := TRUE, 
							Timeout := InTimeout,
							Error => TmpError,
							Busy => TmpBusy,
							ErrorId => TmpErrorId,
						);
					5:
						MB_EL.WriteSingleCoil
						(
							UnitID := InUnitId, 
							Quantity := InQuantity, 
							MBAddr := InStartAddr, 
							cbLength := 2* InQuantity, 
							pMemoryAddr := InAddrDest, 
							Execute := TRUE, 
							Timeout := InTimeout,
							Error => TmpError,
							Busy => TmpBusy,
							ErrorId => TmpErrorId,
						);
					6:
						MB_EL.WriteSingleRegister
						(
							UnitID := InUnitId, 
							Quantity := InQuantity, 
							MBAddr := InStartAddr, 
							cbLength := 2* InQuantity, 
							pMemoryAddr := InAddrDest, 
							Execute := TRUE, 
							Timeout := InTimeout,
							Error => TmpError,
							Busy => TmpBusy,
							ErrorId => TmpErrorId,
						);
					15:
						MB_EL.WriteMultipleCoils
						(
							UnitID := InUnitId, 
							Quantity := InQuantity, 
							MBAddr := InStartAddr, 
							cbLength := 2* InQuantity, 
							pMemoryAddr := InAddrDest, 
							Execute := TRUE, 
							Timeout := InTimeout,
							Error => TmpError,
							Busy => TmpBusy,
							ErrorId => TmpErrorId,
						);
					16:
						MB_EL.WriteRegs
						(
							UnitID := InUnitId, 
							Quantity := InQuantity, 
							MBAddr := InStartAddr, 
							cbLength := 2* InQuantity, 
							pMemoryAddr := InAddrDest, 
							Execute := TRUE, 
							Timeout := InTimeout,
							Error => TmpError,
							Busy => TmpBusy,
							ErrorId => TmpErrorId,
						);
				END_CASE
				
				IF NOT (TmpBusy) AND NOT (TmpError) THEN
					TempoRetry(In:= FALSE);
					TON_ReadRTU(IN:= FALSE ) ; 
					MB_EL.ReadInputRegs(Execute:= FALSE);
					MB_EL.ReadRegs(Execute:= FALSE);
					MB_EL.ReadCoils(Execute:= FALSE);
					MB_EL.ReadInputStatus(Execute:= FALSE);
					MB_EL.WriteSingleCoil(Execute:= FALSE);
					MB_EL.WriteSingleRegister(Execute:= FALSE);
					MB_EL.WriteMultipleCoils(Execute:= FALSE);
					MB_EL.WriteRegs(Execute:= FALSE);
					OutErrorId 		:= 0;
					OutErrorMbRead	:= FALSE;
					AlarmCounter	:= 0; // Reset counter after successful modbus read. 
					OutbCompleted 	:= TRUE ; 
					Step 			:= 0;
					OutBusy         := FALSE;
				ELSIF ((NOT (TmpBusy) AND TmpError) OR TON_ReadRTU.Q)  AND NOT(bRetry) THEN
	
					TempoRetry(In:= FALSE);
					bRetry := FALSE;
					MB_EL.ReadCoils(Execute:= FALSE);
					MB_EL.ReadInputRegs(Execute:= FALSE);
					MB_EL.ReadInputStatus(Execute:= FALSE);
					MB_EL.ReadRegs(Execute:= FALSE);
					MB_EL.WriteSingleCoil(Execute:= FALSE);
					MB_EL.WriteSingleRegister(Execute:= FALSE);
					MB_EL.WriteMultipleCoils(Execute:= FALSE);
					MB_EL.WriteRegs(Execute:= FALSE);
					AlarmCounter 	:= MIN(AlarmCounter + 1,3) ; 
					OutErrorId		:= SEL(TON_ReadRTU.Q , TmpErrorId ,250 );
					Step 			:= 0;
					TON_ReadRTU(IN:= FALSE ) ; 
					OutBusy         := FALSE;
				ELSIF NOT (TmpBusy) AND TmpError AND bRetry THEN
					MB_EL.ReadInputRegs(Execute:= FALSE);
					MB_EL.ReadRegs(Execute:= FALSE);
					MB_EL.ReadCoils(Execute:= FALSE);
					MB_EL.ReadInputStatus(Execute:= FALSE);
					MB_EL.WriteSingleCoil(Execute:= FALSE);
					MB_EL.WriteSingleRegister(Execute:= FALSE);
					MB_EL.WriteMultipleCoils(Execute:= FALSE);
					MB_EL.WriteRegs(Execute:= FALSE);
					step := 2;
					OutBusy         := FALSE;
				END_IF	
			2: 
				TempoRetry(In:= TRUE);		// LEAVE SOME TIME BEFORE NEW ATTEMPT . 
				IF NOT(TempoRetry.Q) THEN
					TempoRetry(In:= FALSE);
					//AlarmCounter := 0;
					step := 0;
					
				END_IF
				
		END_CASE	
	
	

	END_IF

END_FUNCTION_BLOCK

// ---- 00_FunctionsBlocks/Beckhoff/Communication/ModbusRTU/CheckStruct.TcPOU
FUNCTION CheckStruct : BOOL
//Allows to compare 2 Struct_InputRTU, TRUE if struct are the same
VAR_INPUT
	InStruct1 : Struct_InputRTU;
	InStruct2 : Struct_InputRTU;
END_VAR
VAR
	bCompareBuffer 	: BOOL := TRUE;
	KK 				: UINT;
	AdrNull			: Pointer to array[1..125] of word;
END_VAR

IF InStruct1.InBuffer <> adrNull AND instruct2.InBuffer <> AdrNull THEN
	CheckStruct:= MEMCMP(pBuf1 := ADR(instruct1), pBuf2 := ADR(InStruct2), n := SIZEOF(InStruct1)) = 0;

	//FOR KK := 1 TO 125 DO
	//	bCompareBuffer := bCompareBuffer AND (InStruct1.InBuffer^[KK] = InStruct2.InBuffer^[KK]);
	//END_FOR
	//
	//
	//CheckStruct :=(InStruct1.InStartAddr	= InStruct2.InStartAddr	AND InStruct1.InQuantity	= InStruct2.InQuantity	AND InStruct1.InUnitID	    = InStruct2.InUnitID	AND  bCompareBuffer AND InStruct1.InFunction	= InStruct2.InFunction	);
END_IF

END_FUNCTION

// ---- 00_FunctionsBlocks/Beckhoff/DataProcessing/FB_WordsToFloat32MLE.TcPOU
FUNCTION_BLOCK FB_WordsToFloat32MLE
////////////////// 
// Merge two words or one word into a Real with Mid little endian coding.
//Validée par KBT : 8/11/2017 
//////////////////		
VAR_INPUT
	
	InFirstWord AT %MW0: WORD; 		// Word sent or stored first 
	InSecondWord AT %MW1 : WORD; 	// Word sent or stored last  

END_VAR
VAR_OUTPUT
	OutCalReal AT %MD0 : REAL;		//Output : Real
END_VAR

END_FUNCTION_BLOCK

// ---- 01_Equipement_Library/Inverter/FB_INV_Sch4400.TcPOU
FUNCTION_BLOCK FB_INV_Sch4400 EXTENDS FB_INV_Base
// Schneider Conext SmartGen 4400
VAR_INPUT PERSISTENT
	{attribute 'OPC.UA.DA' := '1'} 
	ParamTcpPort					: UINT		:= 502;				(* (NA) TCP port*)
	{attribute 'OPC.UA.DA' := '1'} 
	ParamIPAddress					: STRING; 						(* (NA)Config: IP Adress of PV INverter	*)
	{attribute 'OPC.UA.DA' := '1'} 
	ParamUnitID 					: BYTE; 						(* (NA) Modbus Unit ID *)
	ParamNumInv						: BYTE;             			(* (NA) Number of inverters*)
END_VAR

VAR_INPUT
			MesDataExd		AT %Q*		: INV_Sch4400; 					 // (NA) Inverter Object 
END_VAR

VAR	
	// M_READ VARIABLES//


		FB_ModbusRead	          	: ARRAY[1..9] OF FB_ModbusRead;  // (NA) FB for Modbus Reading
		FB_ModbusWrite				: ARRAY[1..2] OF FB_ModbusWrite;
		AX_ModbusReadAlarm			: ARRAY[1..9] OF BOOL;
		AX_ModbusReadAlarmId		: ARRAY[1..9] OF UDINT;		
		AX_ModbusWriteAlarm			: ARRAY[1..2] OF BOOL;
		AX_ModbusWriteAlarmId		: ARRAY[1..2] OF UDINT;
		
		AX_QTY_MB			: ARRAY[1..2,1..9] OF WORD := [24, 		30, 	10, 	28, 	13, 	2, 		6,		11,2,	24, 	30, 	10, 	28, 	13, 	2, 		6,		11,		2	];
		AX_ADR_MB			: ARRAY[1..2,1..9] OF WORD := [11100, 	11000, 	10401, 	11300, 	11701, 	11600, 	11200,	10500, 11400,	21100, 	21000, 	20401, 	21300, 	21701, 	21600,	21200, 20500, 21400	];
	
		MesBlock1_Temp 				: ARRAY [1..24] OF WORD ; 		// (NA) Temporary Block with multiple modbus reading (Caution : Double Word variables)
		MesBlock2_Temp 				: ARRAY [1..30] OF WORD ; 		// (NA) Temporary Block with multiple modbus reading (Caution : Double Word variables)
		MesBlock3_Temp 				: ARRAY [1..10] OF WORD ; 		// (NA) Temporary Block with multiple modbus reading (Caution : Double Word variables)
		MesBlock4_Temp 				: ARRAY [1..28] OF WORD ; 		// (NA) Temporary Block with multiple modbus reading (Caution : Double Word variables)
		MesBlock5_Temp 				: ARRAY [1..13] OF WORD ; 		// (NA) Temporary Block with multiple modbus reading (Caution : Double Word variables)
		MesBlock6_Temp				: ARRAY [1..2]  OF WORD ;		// (NA) Temporary block with both start commands for each inverter
		MesBlock7_Temp				: ARRAY [1..6]  OF WORD ;		// (NA) 
		MesBlock8_Temp				: ARRAY [1..11] OF WORD ;		// (NA) 
		MesBlock9_Temp				: ARRAY [1..11] OF WORD ;		// (NA) 
		
		MesBlockWrite1_Temp 		: ARRAY[1..4] OF WORD;			// (NA) Temporary Block with multiple modbus writing (Caution : Double Word variables)
		MesBlockWrite2_Temp			: ARRAY[1..2] of WORD;			// (NA) Temporary Block with multiple modbus writing (Caution : Double Word variables)

		TON_BJ						: ARRAY[1..10 ] OF TON ; 

	// M_STARTSTOP//
		StartStop_RTrig				: R_Trig;
              	
	// M_CP
		CalCP_CMD_StartStop			: BOOL; 						// Write command start;
END_VAR

METHOD M_Acknowledge
VAR
		//Each cycle
	Temp_Alarm	:BOOL:=False;	
END_VAR
END_METHOD

METHOD M_AlarmManagement
//////////////////
// Manages IntelliGen Alarms
/////////////////

VAR 
	// Method local variables (reinitialized at each cycle) 
	FB_AlarmCodeManager : FB_AlarmCodeManager ; 
	KK				: BYTE;		// For Loop 
	bComError		: BOOL := TRUE;
	bComWarning 	: BOOL;

	AX_BJHS			: ARRAY[1..10] OF BOOL;
END_VAR
FOR KK := 1 TO 8 DO
	bCOmError := bCOmError AND FB_ModbusRead[KK].ModbusReadAlarm;
	bComWarning := bComWarning OR FB_ModbusRead[KK].ModbusReadAlarm;
END_FOR
bComError := bComError AND FB_ModbusWrite[1].ModbusWriteAlarm AND FB_ModbusWrite[2].ModbusWriteAlarm;
bComWarning := bComError OR FB_ModbusWrite[1].ModbusWriteAlarm OR FB_ModbusWrite[2].ModbusWriteAlarm ;

TON_ComAlarm(IN := bComError, PT := T#30S,Q=> MesDataExd.MesData.MesAlarmCom);
TON_ComWarning(IN := bComWarning, PT := T#30S);

// BJ HS detection 
FOR KK:=1 TO 10 DO 
	TON_BJ[KK]( IN:= MesDataExd.MesData.MesP > 100  AND A1_WS.MesDataExd.MesData.MesGTI > 20 AND MesDataExd.AX_STR[KK].MesIdc < 3 , PT:= T#30S ) ; 
	AX_BJHS[KK] :=  TON_BJ[KK].Q ; 
END_FOR


// ALARM CODE //
	FB_AlarmCodeManager(
		bAlarm1			:= NOT MesDataExd.MesStateCom,		// INV Not Communicating
		bAlarm2			:= FALSE,							// 
		bAlarm3			:= NOT MesDataExd.MesStateCBac,		// INV AC CB opened CB501
		bAlarm4			:= FALSE,							// 	
		bAlarm5			:= NOT MesDataExd.MesStateCBdc,		// INV DC CB opened CB201
		bAlarm6			:= FALSE,							// 
		bAlarm7			:= MesDataExd.MesFaultGnd,			// INV Ground Fault	
		bAlarm8			:= FALSE,							// 
		bAlarm9			:= NOT MesDataExd.MesStateNoAlert, 	// INV has detected an abnormal event which prevents operation
		bAlarm10		:= FALSE, 							// 
		bAlarm11		:= MesDataExd.MesEventID_AbnormalOff > 0,	// ID of the event causing an abnormal stop exists for INV1(not 0)   			#Equipment
		bAlarm12		:= FALSE,							// 
		bAlarm13		:= MesDataExd.MesState <> 23,  		// INV is not in state online PV  									 			#Equipment
		bAlarm14		:= MesDataExd.MesState = 5,			// State Of inverter ID = 5,  Disabled. Inverter is disabled. 		 			#Equipment
		bAlarm15		:= MesDataExd.MesData.MesAlarmCom, 			// No communication frames for the past 30 seconds 					 			#COM
		wAlarmCode		=> MesDataExd.MesData.MesAlarmCode);

// WARNING CODE //
	FB_AlarmCodeManager(
 		bAlarm1			:= MesWarningCom, 							// A frame failed for the last 30s 												#COM
		bAlarm2			:= MesDataExd.MesState = 8,  				// INV is Offline  																#Equipment
		bAlarm3			:= NOT MesDataExd.MesData.MesCP_Read, 	  				// No permission to read from SCADA
		bAlarm4			:= MesDataExd.MesState_TypeSetptP <> 15,	// INV active power setpoint is not MPPT  										#Equipment
		bAlarm5			:= NOT MesDataExd.MesData.MesCP_Write,					// No permission to write from SCADA							
		bAlarm6			:= MesDataExd.MesState_TypeSetptP = 11, 	// INV active power setpoint is limited by communication  						#Equipment	
		bAlarm7			:= MesDataExd.MesState = 20, 				// State Of inverter ID = 20, Lost of production Online var :  Inverter is online in var Mode. AC circuit breaker is closed. #Equipment 
		bAlarm8			:= MesDataExd.MesState_TypeSetptQ = 6 OR  MesDataExd.MesState_TypeSetptQ = 7,   // INV reactive setpoint set by communication   #Equipment
		bAlarm9			:= IN_SetptPlimit_Local < MesDataExd.MesData.ParamPn,  		// INV local active power setpoint is under nominal active power 
		bAlarm10		:= NOT RS_StartStop_Local.Q1,       // Local Stop Command 
		bAlarm11		:= FALSE , //
		bAlarm12		:= FALSE, 							//
		bAlarm13		:= FALSE,							// 
		bAlarm14		:= FALSE,							// 
		bAlarm15		:= FALSE, 							//
		wAlarmCode		=> MesDataExd.MesData.MesWarningCode);	

// EVENT CODE //
	FB_AlarmCodeManager(
		bAlarm1			:= AX_BJHS[1],						// BJ 1 HS  
		bAlarm2			:= AX_BJHS[2],						// BJ 2 HS  
		bAlarm3			:= AX_BJHS[3],						// BJ 3 HS
		bAlarm4			:= AX_BJHS[4],						// BJ 4 HS
		bAlarm5			:= AX_BJHS[5], 						// BJ 5 HS
		bAlarm6			:= AX_BJHS[6], 						// BJ 6 HS
		bAlarm7			:= AX_BJHS[7],						// BJ 7 HS
		bAlarm8			:= AX_BJHS[8],  					// BJ 8 HS
		bAlarm9			:= AX_BJHS[9], 						// BJ 9 HS
		bAlarm10		:= AX_BJHS[10], 					// BJ 10 HS
		bAlarm11		:= NOT RS_StartStop.Q1, 			// Stop command for INV 
		bAlarm12		:= FALSE,  							// 
		bAlarm13		:= FALSE, 							// 
		bAlarm14		:= FALSE, 							// 
		bAlarm15		:= FALSE,							// 		
		wAlarmCode		=>  MesDataExd.MesData.MesEventCode);
END_METHOD

METHOD M_CP
//////////////////
//  Emulator
/////////////////

VAR 
	// Method local variables (reinitialized at each cycle) 
	
END_VAR

	
CalCP_CMD_StartStop	:= FB_ModbusRead[6].OUT_NbRead > 0 AND (MesDataExd.MesStartDisabled  <> NOT  RS_StartStop.Q1);


SUPER^.M_CP() ; 




Trig_Cmd_Read(CLK:=IN_CmdToggleRead);
Trig_Cmd_Write(CLK:=IN_CmdToggleWrite);
	
IF Trig_Cmd_Read.Q THEN
	IN_CmdToggleRead := FALSE;
	MesDataExd.MesData.MesCP_Read := NOT MesDataExd.MesData.MesCP_Read;
END_IF


IF Trig_Cmd_Write.Q THEN
	IN_CmdToggleWrite := FALSE;
	MesDataExd.MesData.MesCP_Write := NOT MesDataExd.MesData.MesCP_Write;
END_IF
END_METHOD

{attribute 'object_name' := 'M_Curtail'}
METHOD M_Curtail
//////////////////
// Write Curtail Command through modbus to PV inverters.  
//////////////////
VAR 
	// Method local variables (reinitialized at each cycle) 

	MW					: FB_MergeWordsToFloat;
	MW_1				: FB_SplitFloatToWords;
	AX_ADR_MB			: ARRAY[1..2] OF  WORD := [11800, 21800];
	AX_QTY_MB			: ARRAY[1..2] OF  BYTE := [4, 4];
	
	InvSetptP_temp		: REAL;
	InvSetptQ_temp		: REAL;
	

	KK: INT;
END_VAR
SUPER^.M_Curtail() ; 
// MODBUS VARIABLE FORMATING //
FB_ModbusWrite[1](WriteCmd := FALSE);
InvSetptP_temp	:= IN_SetptPlimit / MesDataExd.MesData.ParamPn; // MesData.ParamPn;
InvSetptQ_temp	:= IN_SetptQ / MesDataExd.MesData.ParamQn; 

MesDataExd.MesData.OUT_SetptPLimit :=  IN_SetptPlimit ; 
MesDataExd.MesData.OUT_SetptQ :=  IN_SetptQ ; 
		
IF A1_PP.ParamTanPhiCtrl   OR A1_SUBMV.A1_GRID.MesDataExd.OUT_CmdQReg 	THEN	
	MW_1(VAR_IN := InvSetptP_temp,		WORD_STRONG =>  MesBlockWrite1_Temp[2 ], 		WORD_WEAK => MesBlockWrite1_Temp[1 ]);	
	MW_1(VAR_IN := InvSetptQ_temp,		WORD_STRONG =>  MesBlockWrite1_Temp[4 ], 		WORD_WEAK => MesBlockWrite1_Temp[3 ]);	 			
ELSE
	MW_1(VAR_IN := InvSetptP_temp,		WORD_STRONG =>  MesBlockWrite1_Temp[2 ], 		WORD_WEAK => MesBlockWrite1_Temp[1 ]);	
	MesBlockWrite1_Temp[3 ]:= 16#7FC0;
	MesBlockWrite1_Temp[4 ]:= 16#0000;
 
END_IF



FB_ModbusWrite[1]
	(
		pSrcAddr := ADR (MesBlockWrite1_Temp),
		sIPAddr := ParamIPAddress,
		tTimeout := ParamTimeout,
		nMBAddr := AX_ADR_MB[ParamNumInv],
		nTCPport := ParamTCPPort,
		cbLength := SIZEOF(MesBlockWrite1_Temp),
		nQuantity := AX_QTY_MB[ParamNumInv],
		nUnitID := ParamUnitID,
		WriteCmd := ClockWrite AND MesDataExd.MesData.MesCP_Write  ,
		Reset := CmdClearFault_G OR IN_CmdReset_L,
		ErrorId => AX_ModbusWriteAlarmId[1],
		ModbusWriteAlarm => AX_ModbusWriteAlarm[1]
	);
END_METHOD

METHOD M_Execute
//////////////////
//  Method Calls 
/////////////////

VAR 
	// Method local variables (reinitialized at each cycle) 

END_VAR
IF  bInit THEN
	M_Init();
	bInit:= FALSE ; 
ELSIF CmdInit_G THEN 
	bInit:= TRUE ;
END_IF

SUPER^.M_Execute() ;
END_METHOD

METHOD M_Init
VAR_INPUT
END_VAR

VAR
	bCompleted : BOOL := FALSE;
END_VAR
IN_SetptPlimit_Local := ParamPn ; // MesDataExd.MesData.ParamPn ;
END_METHOD

{attribute 'object_name' := 'M_Read'}
METHOD M_Read
//////////
// Read Method for SMA : Modbus reading
//////////
VAR
	// Method local variables (reinitialized at each cycle) 
	MW					: FB_MergeWordsToFloat;
	MW_1				: FB_WordsToDint64BE;
	
	EacInj_Interm1		: ULINT;
	EacCon_Interm1		: ULINT;
	EreacCapa_Interm1	: ULINT;
	EreacInd_Interm1	: ULINT;
	EacInj_Day_Interm1	: ULINT;
	
	EacInj_Interm2		: ULINT;
	EacCon_Interm2		: ULINT;
	EreacCapa_Interm2	: ULINT;
	EreacInd_Interm2	: ULINT;
	EacInj_Day_Interm2	: ULINT;
	
	KK					: BYTE;						 // Index to loop over modbus blocks 	
	JJ					: BYTE;
	
END_VAR
IF MesDataExd.MesData.MesCP_Read THEN		
	
	// MODBUS REQUEST//
		//Electrical Measurements + Ground Measurements
		FB_ModbusRead[1]
		(
			nTCPPort		:= ParamTcpPort,
			ClockRead		:= MesDataExd.MesData.MesCP_Read AND ClockRead, 
			Reset			:= CmdClearFault_G OR IN_CmdReset_L,
			sIPAddr			:=ParamIPAddress ,
			nUnitID			:= 1, 
			tTimeout		:= ParamTimeout,
			nQuantity		:= AX_QTY_MB[ParamUnitID, 1] , 
			nMBAddr			:= AX_ADR_MB[ParamUnitID, 1] , 
			cbLength		:= SIZEOF(MesBlock1_Temp) , 
			pDestAddr		:= ADR(MesBlock1_Temp) , 
			ModbusReadAlarm	=>AX_ModbusReadAlarm[1] , 
			ErrorId			=> AX_ModbusReadAlarmId[1]
		);
			
		//Production Measurements
		FB_ModbusRead[2]
		(
			nTCPPort		:= ParamTcpPort,
			ClockRead		:= MesDataExd.MesData.MesCP_Read AND ClockRead, 
			Reset			:= CmdClearFault_G OR IN_CmdReset_L,
			sIPAddr			:=ParamIPAddress , 
			nUnitID			:= 1, 
			tTimeout		:= ParamTimeout,
			nQuantity		:= AX_QTY_MB[ParamUnitID, 2] , 
			nMBAddr			:= AX_ADR_MB[ParamUnitID, 2] , 
			cbLength		:= SIZEOF(MesBlock2_Temp) , 
			pDestAddr		:= ADR(MesBlock2_Temp) , 
			ModbusReadAlarm	=>AX_ModbusReadAlarm[2] , 
			ErrorId			=> AX_ModbusReadAlarmId[2]
		);
		
		// Status Summary + Event Summary
		FB_ModbusRead[3]
		(
			nTCPPort		:= ParamTcpPort,
			ClockRead		:= MesDataExd.MesData.MesCP_Read AND ClockRead, 
			Reset			:= CmdClearFault_G OR IN_CmdReset_L,
			sIPAddr			:=ParamIPAddress , 
			nUnitID			:= 1, 
			tTimeout		:= ParamTimeout,
			nQuantity		:= AX_QTY_MB[ParamUnitID, 3] , 
			nMBAddr			:= AX_ADR_MB[ParamUnitID, 3] , 
			cbLength		:= SIZEOF(MesBlock3_Temp) , 
			pDestAddr		:= ADR(MesBlock3_Temp) , 
			ModbusReadAlarm	=>AX_ModbusReadAlarm[3] , 
			ErrorId			=> AX_ModbusReadAlarmId[3]
		);
		
		//String Measurements
		FB_ModbusRead[4]
		(
			nTCPPort		:= ParamTcpPort,
			ClockRead		:= MesDataExd.MesData.MesCP_Read AND ClockRead, 
			Reset			:= CmdClearFault_G OR IN_CmdReset_L,
			sIPAddr			:= ParamIPAddress , 
			nUnitID			:= 1, 
			tTimeout		:= ParamTimeout,
			nQuantity		:= AX_QTY_MB[ParamUnitID, 4], 
			nMBAddr			:= AX_ADR_MB[ParamUnitID, 4], 
			cbLength		:= SIZEOF(MesBlock4_Temp), 
			pDestAddr		:= ADR(MesBlock4_Temp), 
			ModbusReadAlarm	=> AX_ModbusReadAlarm[4], 
			ErrorId			=> AX_ModbusReadAlarmId[4]
		);
		
			//Power Commands
		FB_ModbusRead[5]
		(
			nTCPPort		:= ParamTcpPort,
			ClockRead		:= MesDataExd.MesData.MesCP_Read AND ClockRead, 
			Reset			:= CmdClearFault_G OR IN_CmdReset_L,
			sIPAddr			:=ParamIPAddress , 
			nUnitID			:= 1, 
			tTimeout		:= ParamTimeout,
			nQuantity		:= AX_QTY_MB[ParamUnitID, 5] , 
			nMBAddr			:= AX_ADR_MB[ParamUnitID, 5] ,  
			cbLength		:= SIZEOF(MesBlock5_Temp) , 
			pDestAddr		:= ADR(MesBlock5_Temp) , 
			ModbusReadAlarm	=>AX_ModbusReadAlarm[5] , 
			ErrorId			=> AX_ModbusReadAlarmId[5]
		);
		
		FB_ModbusRead[6]
		(
			nTCPPort		:= ParamTcpPort,
			ClockRead		:= MesDataExd.MesData.MesCP_Read AND ClockRead, 
			Reset			:= CmdClearFault_G OR IN_CmdReset_L,
			sIPAddr			:=ParamIPAddress , 
			nUnitID			:= 1, 
			tTimeout		:= ParamTimeout,
			nQuantity		:= AX_QTY_MB[ParamUnitID, 6] , 
			nMBAddr			:= AX_ADR_MB[ParamUnitID, 6] , 
			cbLength		:= SIZEOF(MesBlock6_Temp)  , 
			pDestAddr		:= ADR(MesBlock6_Temp) , 
			ModbusReadAlarm	=> AX_ModbusReadAlarm[6] , 
			ErrorId			=> AX_ModbusReadAlarmId[6]
		);
		
		FB_ModbusRead[7]
		(
			nTCPPort		:= ParamTcpPort,
			ClockRead		:= MesDataExd.MesData.MesCP_Read AND ClockRead, 
			Reset			:= CmdClearFault_G OR IN_CmdReset_L,
			sIPAddr			:=ParamIPAddress , 
			nUnitID			:= 1, 
			tTimeout		:= ParamTimeout,
			nQuantity		:= AX_QTY_MB[ParamUnitID, 7] , 
			nMBAddr			:= AX_ADR_MB[ParamUnitID, 7] , 
			cbLength		:= SIZEOF(MesBlock7_Temp)  , 
			pDestAddr		:= ADR(MesBlock7_Temp) , 
			ModbusReadAlarm	=> AX_ModbusReadAlarm[7] , 
			ErrorId			=> AX_ModbusReadAlarmId[7]
		);
		FB_ModbusRead[8]
		(
			nTCPPort		:= ParamTcpPort,
			ClockRead		:= MesDataExd.MesData.MesCP_Read AND ClockRead, 
			Reset			:= CmdClearFault_G OR IN_CmdReset_L,
			sIPAddr			:=ParamIPAddress , 
			nUnitID			:= 1, 
			tTimeout		:= ParamTimeout,
			nQuantity		:= AX_QTY_MB[ParamUnitID, 8] , 
			nMBAddr			:= AX_ADR_MB[ParamUnitID, 8] , 
			cbLength		:= SIZEOF(MesBlock8_Temp)  , 
			pDestAddr		:= ADR(MesBlock8_Temp) , 
			ModbusReadAlarm	=> AX_ModbusReadAlarm[8] , 
			ErrorId			=> AX_ModbusReadAlarmId[8]
		);	
		
			FB_ModbusRead[9]
		(
			nTCPPort		:= ParamTcpPort,
			ClockRead		:= MesDataExd.MesData.MesCP_Read AND ClockRead, 
			Reset			:= CmdClearFault_G OR IN_CmdReset_L,
			sIPAddr			:=ParamIPAddress , 
			nUnitID			:= 1, 
			tTimeout		:= ParamTimeout,
			nQuantity		:= AX_QTY_MB[ParamUnitID, 9] , 
			nMBAddr			:= AX_ADR_MB[ParamUnitID, 9] , 
			cbLength		:= SIZEOF(MesBlock9_Temp)  , 
			pDestAddr		:= ADR(MesBlock9_Temp) , 
			ModbusReadAlarm	=> AX_ModbusReadAlarm[9] , 
			ErrorId			=> AX_ModbusReadAlarmId[9]
		);	
		
		MW( WORD_STRONG:= MesBlock1_Temp[2  ],	WORD_WEAK := MesBlock1_Temp[1  ], VAR_OUT := MesDataExd.MesI1 );		
		MW( WORD_STRONG:= MesBlock1_Temp[4  ], 	WORD_WEAK := MesBlock1_Temp[3  ], VAR_OUT := MesDataExd.MesI2 );      
		MW( WORD_STRONG:= MesBlock1_Temp[6  ], 	WORD_WEAK := MesBlock1_Temp[5  ], VAR_OUT := MesDataExd.MesI3 );      
		MW( WORD_STRONG:= MesBlock1_Temp[8  ], 	WORD_WEAK := MesBlock1_Temp[7  ], VAR_OUT := MesDataExd.MesV1 );      
		MW( WORD_STRONG:= MesBlock1_Temp[10 ], 	WORD_WEAK := MesBlock1_Temp[9  ], VAR_OUT := MesDataExd.MesV2 );      
		MW( WORD_STRONG:= MesBlock1_Temp[12 ], 	WORD_WEAK := MesBlock1_Temp[11 ], VAR_OUT := MesDataExd.MesV3 );      
		MW( WORD_STRONG:= MesBlock1_Temp[14 ], 	WORD_WEAK := MesBlock1_Temp[13 ], VAR_OUT := MesDataExd.MesData.MesFreq );    
		MW( WORD_STRONG:= MesBlock1_Temp[16 ], 	WORD_WEAK := MesBlock1_Temp[15 ], VAR_OUT := MesDataExd.MesData.MesIdc );     
		MW( WORD_STRONG:= MesBlock1_Temp[18 ], 	WORD_WEAK := MesBlock1_Temp[17 ], VAR_OUT := MesDataExd.MesData.MesUdc );     
		MW( WORD_STRONG:= MesBlock1_Temp[20 ], 	WORD_WEAK := MesBlock1_Temp[19 ], VAR_OUT := MesDataExd.MesU12 );     
		MW( WORD_STRONG:= MesBlock1_Temp[22 ], 	WORD_WEAK := MesBlock1_Temp[21 ], VAR_OUT := MesDataExd.MesU23 );     
		MW( WORD_STRONG:= MesBlock1_Temp[24 ], 	WORD_WEAK := MesBlock1_Temp[23 ], VAR_OUT := MesDataExd.MesU31 );    
			
		MW( WORD_STRONG:= MesBlock2_Temp[2 ], 	WORD_WEAK := 	MesBlock2_Temp[1 ], VAR_OUT := MesDataExd.MesData.MesP );
		MW( WORD_STRONG:= MesBlock2_Temp[4 ], 	WORD_WEAK := 	MesBlock2_Temp[3 ], VAR_OUT := MesDataExd.MesData.MesQ );
		MW_1(InFirstWord := MesBlock2_Temp[7 ], 	InSecondWord := MesBlock2_Temp[8], 	InThirdWord := MesBlock2_Temp[9], 	InFourthWord := MesBlock2_Temp[10], OutCalDint => EacInj_Interm1);
		MW_1(InFirstWord := MesBlock2_Temp[11], 	InSecondWord := MesBlock2_Temp[12], InThirdWord := MesBlock2_Temp[13], 	InFourthWord := MesBlock2_Temp[14], OutCalDint => EacCon_Interm1);
		MW_1(InFirstWord := MesBlock2_Temp[15], 	InSecondWord := MesBlock2_Temp[16], InThirdWord := MesBlock2_Temp[17], 	InFourthWord := MesBlock2_Temp[18], OutCalDint => EreacCapa_Interm1);
		MW_1(InFirstWord := MesBlock2_Temp[19], 	InSecondWord := MesBlock2_Temp[20], InThirdWord := MesBlock2_Temp[21], 	InFourthWord := MesBlock2_Temp[22], OutCalDint => EreacInd_Interm1);
		MW_1(InFirstWord := MesBlock2_Temp[27], 	InSecondWord := MesBlock2_Temp[28], InThirdWord := MesBlock2_Temp[29], 	InFourthWord := MesBlock2_Temp[30], OutCalDint => EacInj_Day_Interm1);
	
		MesDataExd.MesEActProd 					:= ULINT_TO_REAL(EacInj_Interm1)/100;
		MesDataExd.MesEActCons 					:= ULINT_TO_REAL(EacCon_Interm1)/100;
		MesDataExd.MesEReactProd 				:= ULINT_TO_REAL(EreacCapa_Interm1)/100;
		MesDataExd.MesEReactCons 				:= ULINT_TO_REAL(EreacInd_Interm1)/100;
		MesDataExd.MesEday 						:= ULINT_TO_REAL(EacInj_Day_Interm1)/100;
		
		MesDataExd.MesStateCBac					:= WORD_TO_BOOL(MesBlock3_Temp[1]);
		MesDataExd.MesStateCBdc					:= WORD_TO_BOOL(MesBlock3_Temp[2]);
		MesDataExd.MesEarthing_Relay			:= WORD_TO_BOOL(MesBlock3_Temp[3]);
		MesDataExd.MesFaultGnd					:= WORD_TO_BOOL(MesBlock3_Temp[4]);
		MesDataExd.MesStateNoAlert				:= WORD_TO_BOOL(MesBlock3_Temp[5]);
		MesDataExd.MesData.MesState_INV			:= WORD_TO_UINT(MesBlock3_Temp[7]);
		MesDataExd.MesBdrigeCtlMod				:= WORD_TO_UINT(MesBlock3_Temp[8]);
		MesDataExd.MesWorkingHr					:= MesBlock3_Temp[9];	
		
		//MW(WORD_WEAK_F := MesBlock4_Temp[ 1], WORD_STRONG_F := MesBlock4_Temp[ 2], NUMBER_F => MesDataExd.MesSB[1].MesIdc);	
		//MW(WORD_WEAK_F := MesBlock4_Temp[ 3], WORD_STRONG_F := MesBlock4_Temp[ 4], NUMBER_F => MesDataExd.MesSB[2].MesIdc);	
		//MW(WORD_WEAK_F := MesBlock4_Temp[ 5], WORD_STRONG_F := MesBlock4_Temp[ 6], NUMBER_F => MesDataExd.MesSB[3].MesIdc);	
		//MW(WORD_WEAK_F := MesBlock4_Temp[ 7], WORD_STRONG_F := MesBlock4_Temp[ 8], NUMBER_F => MesDataExd.MesSB[4].MesIdc);	
		
		
		IF (ParamNumInv = 1 AND ParamIPAddress = '10.0.0.20') OR (ParamNumInv = 2 AND ParamIPAddress = '10.0.0.30') THEN 
			MW(WORD_WEAK := MesBlock4_Temp[ 9], WORD_STRONG := MesBlock4_Temp[10], VAR_OUT := MesDataExd.AX_STR[10].MesIdc);	
			MW(WORD_WEAK := MesBlock4_Temp[11], WORD_STRONG := MesBlock4_Temp[12], VAR_OUT := MesDataExd.AX_STR[9].MesIdc);	
			MW(WORD_WEAK := MesBlock4_Temp[13], WORD_STRONG := MesBlock4_Temp[14], VAR_OUT := MesDataExd.AX_STR[8].MesIdc);	
			MW(WORD_WEAK := MesBlock4_Temp[15], WORD_STRONG := MesBlock4_Temp[16], VAR_OUT := MesDataExd.AX_STR[7].MesIdc);	
			MW(WORD_WEAK := MesBlock4_Temp[17], WORD_STRONG := MesBlock4_Temp[18], VAR_OUT := MesDataExd.AX_STR[6].MesIdc);	
			MW(WORD_WEAK := MesBlock4_Temp[19], WORD_STRONG := MesBlock4_Temp[20], VAR_OUT := MesDataExd.AX_STR[5].MesIdc);	
			MW(WORD_WEAK := MesBlock4_Temp[21], WORD_STRONG := MesBlock4_Temp[22], VAR_OUT := MesDataExd.AX_STR[4].MesIdc);	
			MW(WORD_WEAK := MesBlock4_Temp[23], WORD_STRONG := MesBlock4_Temp[24], VAR_OUT := MesDataExd.AX_STR[3].MesIdc);	
			MW(WORD_WEAK := MesBlock4_Temp[25], WORD_STRONG := MesBlock4_Temp[26], VAR_OUT := MesDataExd.AX_STR[2].MesIdc);	
			MW(WORD_WEAK := MesBlock4_Temp[27], WORD_STRONG := MesBlock4_Temp[28], VAR_OUT := MesDataExd.AX_STR[1].MesIdc);		
			
		ELSE
			MW(WORD_WEAK := MesBlock4_Temp[ 9], WORD_STRONG := MesBlock4_Temp[10], VAR_OUT := MesDataExd.AX_STR[1].MesIdc);	
			MW(WORD_WEAK := MesBlock4_Temp[11], WORD_STRONG := MesBlock4_Temp[12], VAR_OUT := MesDataExd.AX_STR[2].MesIdc);	
			MW(WORD_WEAK := MesBlock4_Temp[13], WORD_STRONG := MesBlock4_Temp[14], VAR_OUT := MesDataExd.AX_STR[3].MesIdc);	
			MW(WORD_WEAK := MesBlock4_Temp[15], WORD_STRONG := MesBlock4_Temp[16], VAR_OUT := MesDataExd.AX_STR[4].MesIdc);	
			MW(WORD_WEAK := MesBlock4_Temp[17], WORD_STRONG := MesBlock4_Temp[18], VAR_OUT := MesDataExd.AX_STR[5].MesIdc);	
			MW(WORD_WEAK := MesBlock4_Temp[19], WORD_STRONG := MesBlock4_Temp[20], VAR_OUT := MesDataExd.AX_STR[6].MesIdc);	
			MW(WORD_WEAK := MesBlock4_Temp[21], WORD_STRONG := MesBlock4_Temp[22], VAR_OUT := MesDataExd.AX_STR[7].MesIdc);	
			MW(WORD_WEAK := MesBlock4_Temp[23], WORD_STRONG := MesBlock4_Temp[24], VAR_OUT := MesDataExd.AX_STR[8].MesIdc);	
			MW(WORD_WEAK := MesBlock4_Temp[25], WORD_STRONG := MesBlock4_Temp[26], VAR_OUT := MesDataExd.AX_STR[9].MesIdc);	
			MW(WORD_WEAK := MesBlock4_Temp[27], WORD_STRONG := MesBlock4_Temp[28], VAR_OUT := MesDataExd.AX_STR[10].MesIdc);	
		
		END_IF
		
	
		
		// Idc Bj = 461 when no connected . 
		FOR KK:=1 TO 10 DO 
			MesDataExd.AX_STR[KK].MesIdc :=  SEL(MesDataExd.AX_STR[KK].MesIdc>355 , MesDataExd.AX_STR[KK].MesIdc , 0) ; 
		END_FOR
		
	
		MW( WORD_STRONG:= MesBlock5_Temp[2 ],		WORD_WEAK := MesBlock5_Temp[1 ], VAR_OUT := MesDataExd.MesSetptP_CC );		
		MW( WORD_STRONG:= MesBlock5_Temp[4 ],		WORD_WEAK := MesBlock5_Temp[3 ], VAR_OUT := MesDataExd.MesSetptQ_CC );   		
		MW( WORD_STRONG:= MesBlock5_Temp[6 ],		WORD_WEAK := MesBlock5_Temp[5 ], VAR_OUT := MesDataExd.MesSetptCosPhi_CC );  		
		MW( WORD_STRONG:= MesBlock5_Temp[8 ],		WORD_WEAK := MesBlock5_Temp[7 ], VAR_OUT := MesDataExd.ParamTP_RampP );    		
		MW( WORD_STRONG:= MesBlock5_Temp[10],		WORD_WEAK := MesBlock5_Temp[9], VAR_OUT  := MesDataExd.ParamTP_RampQ );    	
		MW( WORD_STRONG:= MesBlock5_Temp[12],		WORD_WEAK := MesBlock5_Temp[11], VAR_OUT := MesDataExd.ParamTP_RampCosPhi ); 	
																								   
		MesDataExd.ParamID_QType 		  := WORD_TO_UINT(MesBlock5_Temp[13]);
		 
		MesDataExd.MesData.MesP			  := MesDataExd.MesData.MesP/1000;
		MesDataExd.MesData.MesQ			  := MesDataExd.MesData.MesQ/1000;
		
		MesDataExd.MesStartDisabled 	  := NOT WORD_TO_BOOL(MesBlock6_Temp[1]);
		MesDataExd.MesStartDisabledPersis := NOT WORD_TO_BOOL(MesBlock6_Temp[2]);
		
		MW( WORD_STRONG:= MesBlock7_Temp[2], 	WORD_WEAK := MesBlock7_Temp[1], VAR_OUT := MesDataExd.MesData.MesI0 );      
		MW( WORD_STRONG:= MesBlock7_Temp[4], 	WORD_WEAK := MesBlock7_Temp[3], VAR_OUT := MesDataExd.MesData.MesInsuResistor );    
		MesDataExd.MesData.MesInsuResistor :=  MesDataExd.MesData.MesInsuResistor / 1000 ; // en kOhms   
		MesDataExd.MesEvendID			  := MesBlock8_Temp[1];
		MesDataExd.MesEventID_Stop		  := MesBlock8_Temp[2];
		MesDataExd.MesStateID_Recovery	  := MesBlock8_Temp[3];
		MesDataExd.MesEventID_AbnormalOff := MesBlock8_Temp[5];
		MesDataExd.MesState_TypeSetptP	  := MesBlock8_Temp[6];
		MW(WORD_WEAK := MesBlock8_Temp[7], WORD_STRONG := MesBlock8_Temp[8], VAR_OUT:= MesDataExd.MesSetptP);
		MesDataExd.MesState_TypeSetptQ	  := MesBlock8_Temp[9];
		MW(WORD_WEAK := MesBlock8_Temp[10], WORD_STRONG := MesBlock8_Temp[11], VAR_OUT := MesDataExd.MesSetptQ);
	
		MW(WORD_WEAK := MesBlock9_Temp[ 1], WORD_STRONG := MesBlock9_Temp[ 2], VAR_OUT := MesDataExd.MesTempExt);	
		// Evaluate 
		MesDataExd.MesData.MesPdc		:=  MesDataExd.MesData.MesIdc * MesDataExd.MesData.MesUdc ;
		MesDataExd.MesData.MesI			:= (MesDataExd.MesI1 + MesDataExd.MesI2 + MesDataExd.MesI3) /3;
		MesDataExd.MesData.MesU			:= (MesDataExd.MesU12 + MesDataExd.MesU23 + MesdataExd.MesU31) /3 ; 
		MesDataExd.MesData.MesV 		:= (MesDataExd.MesV1 + MesDataExd.MesV2 + MesdataExd.MesV3) /3 ; 
		MesDataExd.MesData.MesS			:= SQRT(MesDataExd.MesData.MesP*MesDataExd.MesData.MesP + MesDataExd.MesData.MesQ* MesDataExd.MesData.MesQ); 
	
		MesDataExd.MesData.MesAlarmCom  := TON_ComAlarm.Q; 
		MesDataExd.MesStateCom 			:= NOT MesDataExd.MesData.MesAlarmCom; 
	
		//MesData 						:= MesDataExd.MesData; 
		
		// Evaluate 
		MesDataExd.MesData.MesPdc	:= MesDataExd.MesData.MesIdc * MesDataExd.MesData.MesUdc ;
		MesDataExd.MesData.MesI					:= (MesDataExd.MesI1 + MesDataExd.MesI2 + MesDataExd.MesI3) /3;
		MesDataExd.MesData.MesU	:= (MesDataExd.MesU12 + MesDataExd.MesU23 + MesdataExd.MesU31) /3 ; 
		MesDataExd.MesData.MesV 	:= (MesDataExd.MesV1 + MesDataExd.MesV2 + MesdataExd.MesV3) /3 ; 
		MesDataExd.MesData.MesS	:= SQRT(MesDataExd.MesData.MesP*MesDataExd.MesData.MesP + MesDataExd.MesData.MesQ* MesDataExd.MesData.MesQ  ) ; 
		//MesData.MesTemp	:= ;   unavailable . 
		//MesData.MesIDState	:= ; Unavaialable . 
		//MesData.MesPF := ; Unavailable . 
		MesDataExd.MesData.ParamPn := ParamPn ; 
		MesDataExd.MesData.MesAlarmCom	:= TON_ComAlarm.Q  ; 
		MesDataExd.MesStateCom := NOT MesDataExd.MesData.MesAlarmCom ; 
		//MesData. CalCurtailing := IN_SetptPlimit < ParamPnom *0.9  ; 
		
END_IF

	
	MesDataExd.MesData.ParamPn 		:= ParamPn ; 
	MesDataExd.MesData.ParamQn 		:= ParamQn ;
END_METHOD

METHOD M_StartStop
VAR
	KK : UINT;
	AX_ADR_MB			: ARRAY[1..2] OF WORD := [11600, 21600];
	AX_QTY_MB			: ARRAY[1..2] OF BYTE := [2, 2];
	
END_VAR
SUPER^.M_StartStop(); 

Trig_Local_Start(CLK:=IN_CmdStart_Local);
Trig_Local_Stop(CLK:=IN_CmdStop_Local);
Trig_Start(CLK:=IN_CmdStart);
Trig_Stop(CLK:=IN_CmdStop);

//RS_StartStop_Local(SET:=Trig_Local_Start.Q,Reset1:= Trig_Local_Stop.Q); // TRUE START, FALSE STOP
//RS_StartStop(SET:=Trig_Start.Q,Reset1 := Trig_Stop.Q); // TRUE START, FALSE STOP
IF Trig_Local_Start.Q OR Trig_Local_Stop.Q OR Trig_Stop.Q OR Trig_Start.Q THEN
	RS_StartStop(SET:=(IN_CmdStart_Local AND NOT IN_CmdStop_Local) OR (IN_CmdStart AND NOT (IN_CmdStop OR IN_CmdStop_Local)), 
			 Reset1 := IN_CmdStop_Local OR (IN_CmdStop AND NOT IN_CmdStart_Local)); 
END_IF

FB_ModbusWrite[2](WriteCmd := FALSE);

//Read the setpoints
	// Evaluate the cmd given 

	MesBlockWrite2_Temp[1] := BOOL_TO_WORD(RS_StartStop.Q1);
	MesBlockWrite2_Temp[2] := BOOL_TO_WORD(RS_StartStop.Q1);
	
	
	MesDataExd.MesData.OUT_CmdStart := RS_StartStop.Q1 ; 
	MesDataExd.MesData.OUT_CmdStop  := NOT RS_StartStop.Q1 ; 	
	
	StartStop_RTrig(CLK:=CalCP_CMD_StartStop);
	
	FB_ModbusWrite[2]
	(
		pSrcAddr := ADR (MesBlockWrite2_Temp),
		sIPAddr := ParamIPAddress,
		tTimeout := ParamTimeout,
		nMBAddr := AX_ADR_MB[ParamUnitID],
		nTCPport := ParamTCPPort,
		cbLength := SIZEOF(MesBlockWrite2_Temp),
		nQuantity := AX_QTY_MB[ParamUnitID],
		nUnitID := ParamUnitID,
		WriteCmd := StartStop_RTrig.Q AND MesDataExd.MesData.MesCP_Write ,
		Reset := CmdClearFault_G,
		ErrorId => AX_ModbusWriteAlarmId[2],
		ModbusWriteAlarm => AX_ModbusWriteAlarm[2]
	);
	
SUPER^.M_Curtail() ;
END_METHOD

METHOD M_StateManager
//////////////////
// Detect which is the state of the inverter. IF loss of communication MesState =0 , the last inverter state is kept .  
/////////////////

VAR 
	// Method local variables (reinitialized at each cycle) 

	
END_VAR
//O=Stopped, 1 = MPPT, 2 = Sleeping, 3 = Starting, 4 = Throttled, 5 = Shutting down, 6 = Fault, 7 = Standby

MesDataExd.MesData.MesState 			:= 0  ; 

//Stopped
	IF MesDataExd.MesData.MesState_INV = 0 OR MesDataExd.MesData.MesState_INV = 5 OR MesDataExd.MesData.MesState_INV = 8 THEN 
		MesDataExd.MesData.MesState.0 := 1;

//MPPT
	ELSIF MesDataExd.MesData.MesState_INV = 23 OR MesDataExd.MesData.MesState_INV = 20 OR MesDataExd.MesData.MesState_INV = 21  OR MesDataExd.MesData.MesState_INV = 25 THEN
			MesDataExd.MesData.MesState.1 := 1;

//Sleeping
//	ELSIF MesDataExd.MesData.MesState_INV = 23 THEN
//			MesDataExd.MesData.MesState.2 := 1;

//Starting		
	ELSIF MesDataExd.MesData.MesState_INV = 12 OR MesDataExd.MesData.MesState_INV = 13 OR MesDataExd.MesData.MesState_INV = 14 OR MesDataExd.MesData.MesState_INV = 15 OR MesDataExd.MesData.MesState_INV = 19 THEN
			MesDataExd.MesData.MesState.3 := 1;

////throttled		
//	ELSIF MesDataExd.MesData.MesState_INV = 23 THEN
//			MesDataExd.MesData.MesState.4 := 1;	

//Shutting down		
	ELSIF MesDataExd.MesData.MesState_INV = 11 THEN
			MesDataExd.MesData.MesState.5 := 1;	

//fault		
	ELSIF MesDataExd.MesData.MesState_INV = 23 THEN
			MesDataExd.MesData.MesState.6 := 1;	

//Standby		
	ELSIF MesDataExd.MesData.MesState_INV = 2 OR MesDataExd.MesData.MesState_INV = 3 OR MesDataExd.MesData.MesState_INV = 18 THEN
			MesDataExd.MesData.MesState.7 := 1;	
	END_IF

SUPER^.M_StateManager() ;
END_METHOD

END_FUNCTION_BLOCK

// ---- 00_FunctionsBlocks/Beckhoff/DataProcessing/FB_MergeWordsToFloat.TcPOU
FUNCTION_BLOCK FB_MergeWordsToFloat
////////////////// 
// Merge two words into a real with IEEE 754 coding (for float reading). 
//////////////////	
VAR_IN_OUT
	VAR_OUT 		 			 : REAL;	
END_VAR


VAR_INPUT
	WORD_STRONG 		AT %MB82 : WORD; // Strong Word 
	WORD_WEAK 			AT %MB80 : WORD; // Weak Word. 
END_VAR

VAR_OUTPUT
	OUT_NanError			: BOOL ; 
END_VAR

VAR
	NUMBER_F_OLD		AT %MB80	: REAL; 	// Works only if the Fb is instantied once per call in the Fb and not the Methods.
	
END_VAR

IF NOT(NUMBER_F_OLD = NUMBER_F_OLD) THEN
	OUT_NanError := TRUE ; 
ELSE
	VAR_OUT :=  NUMBER_F_OLD ; 
	OUT_NanError := FALSE ; 
END_IF

END_FUNCTION_BLOCK

// ---- 00_FunctionsBlocks/Beckhoff/DataProcessing/FB_SplitFloatToWords.TcPOU
FUNCTION_BLOCK FB_SplitFloatToWords
////////////////// 
// Merge two words into a real with IEEE 754 coding (for float reading). 
//////////////////	
VAR_INPUT
	
	VAR_IN 		AT %MD0 : REAL;
END_VAR

VAR_OUTPUT
	
	WORD_STRONG 	AT %MW1 : WORD; // Strong Word 
	WORD_WEAK 	AT %MW0 : WORD; // Weak Word. 
END_VAR

END_FUNCTION_BLOCK

// ---- 00_FunctionsBlocks/Common/DataProcessing/MergeWord/FB_WordsToDint64BE.TcPOU
FUNCTION_BLOCK FB_WordsToDint64BE
////////////////// 
// Merge four words into a DINT or UDINT with big endian coding. And finally Output a Real. 
//////////////////	
VAR_OUTPUT
	OutCalDint : ULINT ; 	
END_VAR

VAR_INPUT
	InFirstWord 		: WORD; 
	InSecondWord 		: WORD; 
	InThirdWord 		: WORD; 
	InFourthWord 		: WORD; 
END_VAR

OutCalDint:= LWORD_TO_ULINT( (SHL(WORD_TO_LWORD(InFirstWord),48) OR SHL(WORD_TO_LWORD(InFirstWord),32)OR SHL(WORD_TO_LWORD(InThirdWord),16)OR WORD_TO_LWORD(InFourthWord)));

END_FUNCTION_BLOCK

// ---- 01_Equipement_Library/Inverter/FB_INV_SmaSCXXXXCP_HE.TcPOU
FUNCTION_BLOCK FB_INV_SmaSCXXXXCP_HE EXTENDS FB_INV_Base

// SMA Sunny Central CP series
VAR_INPUT PERSISTENT
	{attribute 'OPC.UA.DA' := '1'} 
	ParamTcpPort				: UINT	:= 502 ;	(* Modbus TCP port							*)	
	
	{attribute 'OPC.UA.DA' := '1'}                
	ParamIPAddress				: STRING; 			(* (NA)Config: IP Adress of PV INverter	    *)
	{attribute 'OPC.UA.DA' := '1'}                  
	ParamUnitID 				: BYTE; 			(* (NA)   SMA Modbus Unit ID.               *)
	ParamNumInv					: BYTE;             (* Inverter Index                           *)
END_VAR

VAR_INPUT 
	// Parameters of the Object (instance specific) 
	AcknowledgeOrder			: BOOL ;			(* Acknowledge fault										*)
	ParamNbInv					: WORD ;			(* (NA) Nb of inverters per inverter                        *)
	                                               
	ParamOptionActivated		: WORD ;			(* (NA) Option available on the inverter                    *)
	                                             
	ParamPRamp					:  REAL:= 0 ;		(* (s) duration of the ramp from setpoint to setpoint       *)
	ParamQRamp					:  REAL:= 0 ;		(* (s) duration of the ramp from setpoint to setpoint       *)
	ParamPfRamp					:  REAL:= 0 ;		(* (s) duration of the ramp from setpoint to setpoint       *)
                                                                                                                
	IN_MesAcCbOpen_IO			:  BOOL ; 			(* Retour cablé Physique des contacteur AC des onduleurs	*)
	Cmd_SwitchOff				:  BOOL ;		    (* etat de DO cablé sur les onduleurs pour les eteindres    *)
	
	
		MesDataExd		AT %Q*	: INV_SmaSCXXXCP_HE;
	
END_VAR



VAR
	//M_Acknowledge
		
	// M_ALARMMNGMT VARIABLES //
	
	
	// M_READ VARIABLES//

		///MesDataExd.MesData.C_Read				:  INV_CC;	
		///MesDataExd.MesData.C_Cmd				:  INV_CC;
		
	
		FB_ModbusRead	          	: ARRAY[1..8] OF FB_ModbusRead; 	            // (NA) FB for Modbus Reading
		FB_ModbusWrite				: ARRAY[1..3] OF FB_ModbusWrite;
		AX_ModbusReadAlarm			: ARRAY[1..9] OF BOOL;
		AX_ModbusReadAlarmId		: ARRAY[1..9] OF UDINT;		
		AX_ModbusWriteAlarm			: ARRAY[1..3] OF BOOL;
		AX_ModbusWriteAlarmId		: ARRAY[1..3] OF UDINT;
		
		
		BlockInit					: WORD;							// First Block : Number of inverters in the PCS
		MesBlock1_Temp 				: ARRAY [1..70] OF WORD ; 		// (NA) Temporary Block with multiple modbus reading (Caution : Double Word variables)
		MesBlock2_Temp 				: ARRAY [1..90] OF WORD ; 		// (NA) Temporary Block with multiple modbus reading (Caution : Double Word variables)
		MesBlock3_Temp 				: ARRAY [1..74] OF WORD ; 		// (NA) Temporary Block with multiple modbus reading (Caution : Double Word variables)
		MesBlock4_Temp 				: ARRAY [1..38] OF WORD ; 		// (NA) Temporary Block with multiple modbus reading (Caution : Double Word variables)
		MesBlock5_Temp 				: ARRAY [1..28] OF WORD ; 		// (NA) Temporary Block with multiple modbus reading (Caution : Double Word variables)
		MesBlock6_Temp				: ARRAY [1..13] OF WORD ;		// (NA) Temporary block with both start commands for each inverter
		MesBlock7_Temp				: ARRAY [1..16] OF WORD ;	
		MesBlock8_Temp				: ARRAY [1..4] OF WORD ;
		
		MesBlockWrite1_Temp 		: WORD ;				    	// (NA) Temporary Block with multiple modbus writing (Caution : Double Word variables)
		MesBlockWrite2_Temp			: WORD ;						// (NA) Temporary Block with multiple modbus writing (Caution : Double Word variables)
		MesBlockWrite3_Temp			: ARRAY [1..2] OF WORD ;
	// M_CURTAIL VARIABLES //
	
		LastCurtailMode				: BOOL:=TRUE ;				// Init at true, to force the first write on inverter
		MesCP_WriteCurtailMode		: BOOL ;
		CurtailModeValue_P			: DWORD ; 					// 1077 := WctlMan : Inverter set setpoint, 1079 := WCtlCom Inverter take the setpoint set by com (plc),303 := OFF
		CurtailModeValue_Q			: DWORD ;					// 303:=OFF,1075:= PFCtlCom,1074:= PFCtlMan,1072 VarCtlCom
		
		MesModbusWriteCode          : UDINT ; 					// (NA) Modbus Write Alarm Code 	
		MesModbusCurtailAlarm		: BOOL ;				   	// (NA) Modbus Write Curtail Alarm 
		
		InvQModeValue				: UINT ;					// Mode of Q power control : 1: Q mod, 2: PF mode, 3: Q(P)
		InvSetptQ					: REAL ;					// (kVAr) setpoint for the reactive power for each inverter
		
	
		InvSetptP					: REAL ;					// (kW) Setpoint for the active power for each inverter
		TEMP						: BOOL ;
	// M_INIT //
		Code_Ctrl_Com 				: UINT := 1079 ;
		
		MesModbusCurtailInitAlarm 	: BOOL ;
		
	// M_STARTSTOP//
		StartStop_RTrig				: R_Trig ;
		StartStop_RTrigIO			: R_Trig ;
		
	// M_CP
		CalCP_Acknowledge			: BOOL ;
		//CalCP_CMD_SetPt				: BOOL; 	  // Write command start;
		CalCP_CMD_StartStop			: BOOL ; 		  // Write command start;
		CalCP_CMD_StartStopIO		: BOOL ; 		  // Write command start;
	// M_STATEMANAGER//
	
	//M_EXECUTE VARIABLES //
		TP_READ						: LTP ;			  //Tempo de cadencement FB Modbus
		RTrig						: R_Trig ; 		  //Front montant sur TP_READ.Q
		ReadBusy					: BOOL ;		 //FB Modbus en busy
		
	//EMULATOR VARIABLES //
		
END_VAR

METHOD M_AlarmManagement
//////////////////
// Manages IntelliGen Alarms
/////////////////

VAR 
	// Method local variables (reinitialized at each cycle) 
	FB_AlarmCodeManager : FB_AlarmCodeManager ; 
	KK				: BYTE;		// For Loop 
	bComError		: BOOL := TRUE;
	bComWarning 	: BOOL;
	AC_CB_OPEN		: BOOL;
END_VAR
FOR KK := 1 TO 6 DO
	bCOmError := bCOmError AND FB_ModbusRead[KK].ModbusReadAlarm;
	bComWarning := bComWarning OR FB_ModbusRead[KK].ModbusReadAlarm;
END_FOR
bComError := bComError AND FB_ModbusWrite[1].ModbusWriteAlarm AND FB_ModbusWrite[2].ModbusWriteAlarm;
bComWarning := bComError OR FB_ModbusWrite[1].ModbusWriteAlarm OR FB_ModbusWrite[2].ModbusWriteAlarm ;

TON_ComAlarm(IN := bComError, PT := T#30S , Q=> MesDataExd.Mesdata.MesAlarmCom);
TON_ComWarning(IN := bComWarning, PT := T#30S);
AC_CB_OPEN := IN_MesAcCbOpen_IO; //  MesDataExd.MesData.MesOpened_CBac OR MesAcCbOpen_IO;


// ALARM CODE //
	FB_AlarmCodeManager(
		bAlarm1			:= MesDataExd.MesState_Inv = 1392	, 	//Inverter in error  #Equipment
		bAlarm2			:= MesDataExd.MesState_Inv = 381,		// INV in stopped mode  #Equipment
		bAlarm3			:= MesDataExd.MesOpened_CBac,			// INV1 AC CB opened CB501
		bAlarm4			:= MesDataExd.MesState_KeyComut, 			// Commateur clef face avant ou DO branché sur onduleur
		bAlarm5			:= MesDataExd.MesOpened_CBdc,				// INV1 DC CB opened CB201
		bAlarm6			:= MesDataExd.MesOpened_CBGrid,			// GridContactor open
		bAlarm7			:= MesDataExd.MesOpened_GFDI	,		// INV1 Ground Fault	
		bAlarm8			:= OUT_Cmd_SwitchOff_IO,						// Commande stop par IO.
		bAlarm9			:= IN_MesAcCbOpen_IO	,					// Etat ac cb IO
		bAlarm10		:= FALSE , 							// 
		bAlarm11		:= FALSE,								// 
		bAlarm12		:= FALSE,								// 
		bAlarm13		:= FALSE,  								//
		bAlarm14		:= FALSE,								// 
		bAlarm15		:= TON_ComAlarm.Q, 						// No communication frames for the past 30 seconds #COM
		wAlarmCode		=>MesDataExd.MesData.MesAlarmCode);

// WARNING CODE //
	FB_AlarmCodeManager(
 		bAlarm1			:= FALSE, 													// 
		bAlarm2			:= MesDataExd.MesState_Inv = 455,  								// INV1 in warning  #Equipment
		bAlarm3			:= NOT MesDataExd.MesData.MesCP_Read, 	  							// Pas le droit en Lecture depuis scada
		bAlarm4			:= FALSE,															// 
		bAlarm5			:= NOT MesDataExd.MesData.MesCP_Write,								// Pas le droit d'ecriture depuis Scada						
		bAlarm6			:= FALSE , 															// 
		bAlarm7			:= FALSE, 															// 
		bAlarm8			:= FALSE, 															//
		bAlarm9			:= IN_SetptPlimit_Local < ParamPn, 								// Onduleur en ecretage par Scada
		bAlarm10		:= NOT RS_StartStop_Local.Q1,                  						// Local Stop Command, 
		bAlarm11		:= FALSE, //
		bAlarm12		:= FALSE, //
		bAlarm13		:= FALSE, //
		bAlarm14		:= FALSE, //
		bAlarm15		:= TON_ComWarning.Q, 												//One or more than error, communication frames for the past 30 seconds #COM
		wAlarmCode		=>MesDataExd.MesData.MesWarningCode);	

// EVENT CODE //
	FB_AlarmCodeManager(
		bAlarm1			:= FALSE, 								// 
		bAlarm2			:= FALSE,								//
		bAlarm3			:= FALSE,								//	
		bAlarm4			:= FALSE,								// 
		bAlarm5			:= FALSE,								// 
		bAlarm6			:= FALSE, 								// 
		bAlarm7			:= NOT RS_StartStop.Q1, 				// Stop command for INV1
		bAlarm8			:= FALSE,  								// 
		bAlarm9			:= FALSE,  								//  
		bAlarm10		:= FALSE,  								//  
		bAlarm11		:= FALSE,   							// 
		bAlarm12		:= FALSE,   							// 
		bAlarm13		:= FALSE,   							// 
		bAlarm14		:= FALSE,  								//  
		bAlarm15		:= FALSE,  								//  
		wAlarmCode		=>MesDataExd.MesData.MesEventCode);
END_METHOD

METHOD M_CP
//////////////////
//  Emulator
/////////////////

VAR 
	// Method local variables (reinitialized at each cycle) 
	MesOpState : BOOL;
END_VAR
//Si une valeur de consigne change alors on ecrit les registres
SUPER^.M_CP() ; 


IF MesDataExd.MesState_Inv = 381 OR MesDataExd.MesState_Inv = 1560  THEN  //STOP
 	MesOpState := 0;
END_IF;
	

RS_StartStop_Local(SET:=IN_CmdStart_Local,Reset1:= IN_CmdStop_Local); // TRUE START, FALSE STOP
RS_StartStop(SET:=IN_CmdStart ,Reset1 := IN_CmdStop OR NOT RS_StartStop_Local.Q1 ); // TRUE START, FALSE STOP



CalCP_CMD_StartStop	:= MesDataExd.MesOpStateOn <>  RS_StartStop.Q1; //FB_ModbusRead[6].OUT_NbRead > 0 AND (MesOpState  =  RS_StartStop.Q1);
CalCP_CMD_StartStopIO	:= MesOpState <>  NOT RS_StartStop.Q1;






Trig_Cmd_Read(CLK:=IN_CmdToggleRead);
Trig_Cmd_Write(CLK:=IN_CmdToggleWrite);
	
IF Trig_Cmd_Read.Q THEN
	IN_CmdToggleRead := FALSE;
	MesDataExd.MesData.MesCP_Read := NOT MesDataExd.MesData.MesCP_Read;
END_IF


IF Trig_Cmd_Write.Q THEN
	IN_CmdToggleWrite := FALSE;
	MesDataExd.MesData.MesCP_Write := NOT MesDataExd.MesData.MesCP_Write;
END_IF
END_METHOD

{attribute 'object_name' := 'M_Curtail'}
METHOD M_Curtail
//////////////////
// Write Curtail Command through modbus to PV inverters.  
//////////////////
VAR 
	// Method local variables (reinitialized at each cycle) 

	AX_ADR_MB			: WORD := 40022;
	AX_QTY_MB			: BYTE := 2;
	AX_UnitID_MB		: BYTE := 2;
	
	InvSetptP_temp		: WORD;
	InvSetptQ_temp		: WORD;
	

	KK: INT;
END_VAR
SUPER^.M_Curtail() ; 
// MODBUS VARIABLE FORMATING //
FB_ModbusWrite[1](WriteCmd := FALSE);


IF MesDataExd.MesData.MesState_Inv.0 THEN 	// Si onduleur est a l'arrêt , on envoi une comamnde non nulle, pour ne pas bloquer son redémarrage
	IN_SetptPlimit := 50 ;
END_IF


InvSetptP_temp	:= REAL_TO_WORD(IN_SetptPlimit*100 / ParamPn)*100;
InvSetptQ_temp	:= REAL_TO_WORD(IN_SetptQ*100 / ParamPn)*100;

		
IF A1_PP.ParamTanPhiCtrl  OR A1_SUBMV.A1_GRID.MesDataExd.OUT_CmdQReg	THEN	
	MesBlockWrite2_Temp	:= InvSetptQ_temp;
	MesBlockWrite1_Temp	:= InvSetptP_temp;
ELSE
	MesBlockWrite1_Temp:= InvSetptP_temp;
	MesBlockWrite2_Temp:= 0;
 
END_IF

FB_ModbusWrite[1]
(
	pSrcAddr := ADR (MesBlockWrite1_Temp),
	sIPAddr := ParamIPAddress,
	tTimeout := ParamTimeout,
	nMBAddr := 40023,
	nTCPport := ParamTCPPort,
	cbLength := SIZEOF(MesBlockWrite1_Temp),
	nQuantity := 1,
	nUnitID := 2,
	WriteCmd := ClockWrite AND MesDataExd.Mesdata.MesCP_Write  ,
	Reset := CmdClearFault_G OR IN_CmdReset_L,
	ErrorId => AX_ModbusWriteAlarmId[1],
	ModbusWriteAlarm => AX_ModbusWriteAlarm[1]
);

	FB_ModbusWrite[2]
(
	pSrcAddr := ADR (MesBlockWrite2_Temp),
	sIPAddr := ParamIPAddress,
	tTimeout := ParamTimeout,
	nMBAddr := 40022,
	nTCPport := ParamTCPPort,
	cbLength := SIZEOF(MesBlockWrite2_Temp),
	nQuantity := 1,
	nUnitID := 2,
	WriteCmd := ClockWrite AND MesDataExd.Mesdata.MesCP_Write  ,
	Reset := CmdClearFault_G OR IN_CmdReset_L,
	ErrorId => AX_ModbusWriteAlarmId[2],
	ModbusWriteAlarm => AX_ModbusWriteAlarm[2]
);
END_METHOD

METHOD M_Execute
//////////////////
//  Method Calls 
/////////////////

VAR 
	// Method local variables (reinitialized at each cycle) 

END_VAR
IF  bInit THEN
	M_Init();
END_IF


SUPER^.M_Execute() ;
END_METHOD

METHOD M_Init
VAR_INPUT
END_VAR

VAR
	bCompleted : BOOL := FALSE;
END_VAR
ParamPn := 1100;
ParamQn := 1100;

IN_SetptPlimit_Local := ParamPn ;
RS_StartStop_Local(Set:= TRUE);
RS_StartStop_Local(Set:= FALSE);

bInit := FAlse;
END_METHOD

{attribute 'object_name' := 'M_Read'}
METHOD M_Read
//////////
// Read Method for SMA : Modbus reading
//////////
VAR
	// Method local variables (reinitialized at each cycle) 
	//MW					: FB_MergeWordsToFloat;
	//MW_1				: FB_WordsToDint64BE;
	

	MW					: FB_MergeWordsToDint;
	AX_QTY_MB			: ARRAY[1..8] OF WORD := [70,	90, 	74, 	38, 	28, 	13,			16,			4		];
	AX_ADR_MB			: ARRAY[1..8] OF WORD := [30197,30533, 	30769, 	34109, 	34613, 	40009,		31793,		32053	];
	AX_UnitID			: ARRAY[1..8] OF BYTE := [3, 	3,		3,		3, 		3,		3,			4,			4		];
	TimeInterm			: REAL;
	
	ID_SSM				: BYTE := 1 ; 
	
	PosInterm			: REAL;
	IdcTotal			: REAL;	
	KK: BYTE;
END_VAR
IF MesDataExd.MesData.MesCP_Read THEN		


	// MODBUS REQUEST//
	//Electrical Measurements + Ground Measurements
	
	FB_ModbusRead[1]
	(
		nTCPPort	:= ParamTcpPort,
		ClockRead:= MesDataExd.MesData.MesCP_Read AND ClockRead, 
		Reset:= CmdClearFault_G OR IN_CmdReset_L,
		sIPAddr:=ParamIPAddress ,
		nUnitID:= AX_UnitID[1], 
		tTimeout:= ParamTimeout,
		nQuantity		:= AX_QTY_MB[1] , 
		nMBAddr			:= AX_ADR_MB[1] , 
		cbLength		:= SIZEOF(MesBlock1_Temp) , 
		pDestAddr		:= ADR(MesBlock1_Temp) , 
		ModbusReadAlarm	=>AX_ModbusReadAlarm[1] , 
		ErrorId			=> AX_ModbusReadAlarmId[1]
	);
	
(* NOT AVAIL FOR THIS INVERTER 
	//Production Measurements
	FB_ModbusRead[2]
	(
		nTCPPort	:= ParamTcpPort,
		ClockRead:= MesDataExd.MesData.MesCP_Read AND ClockRead, 
		Reset:= CmdClearFault_G OR IN_CmdReset_L,
		sIPAddr:=ParamIPAddress , 
		nUnitID:= AX_UnitID[2], 
		tTimeout:= ParamTimeout,
		nQuantity		:= AX_QTY_MB[2] , 
		nMBAddr			:= AX_ADR_MB[2] , 
		cbLength		:= SIZEOF(MesBlock2_Temp) , 
		pDestAddr		:= ADR(MesBlock2_Temp) , 
		ModbusReadAlarm	=>AX_ModbusReadAlarm[2] , 
		ErrorId			=> AX_ModbusReadAlarmId[2]
	);
	
	*) 
	
	// Status Summary + Event Summary
	FB_ModbusRead[3]
	(
		nTCPPort	:= ParamTcpPort,
		ClockRead:= MesDataExd.MesData.MesCP_Read AND ClockRead, 
		Reset:= CmdClearFault_G OR IN_CmdReset_L,
		sIPAddr:=ParamIPAddress , 
		nUnitID:= AX_UnitID[3], 
		tTimeout:= ParamTimeout,
		nQuantity		:= AX_QTY_MB[3] , 
		nMBAddr			:= AX_ADR_MB[3] , 
		cbLength		:= SIZEOF(MesBlock3_Temp) , 
		pDestAddr		:= ADR(MesBlock3_Temp) , 
		ModbusReadAlarm	=>AX_ModbusReadAlarm[3] , 
		ErrorId			=> AX_ModbusReadAlarmId[3]
	);
	
	
	//String Measurements
	FB_ModbusRead[4]
	(
		nTCPPort	:= ParamTcpPort,
		ClockRead:= MesDataExd.MesData.MesCP_Read AND ClockRead, 
		Reset:= CmdClearFault_G OR IN_CmdReset_L,
		sIPAddr:=ParamIPAddress , 
		nUnitID:= AX_UnitID[4], 
		tTimeout:= ParamTimeout,
		nQuantity		:= AX_QTY_MB[4] , 
		nMBAddr			:= AX_ADR_MB[4] , 
		cbLength		:= SIZEOF(MesBlock4_Temp) , 
		pDestAddr		:= ADR(MesBlock4_Temp) , 
		ModbusReadAlarm	=>AX_ModbusReadAlarm[4] , 
		ErrorId			=> AX_ModbusReadAlarmId[4]
	);
	

(* not available for this inverter 
		//Power Commands
	FB_ModbusRead[5]
	(
		nTCPPort	:= ParamTcpPort,
		ClockRead:= MesDataExd.MesData.MesCP_Read AND ClockRead, 
		Reset:= CmdClearFault_G OR IN_CmdReset_L,
		sIPAddr:=ParamIPAddress , 
		nUnitID:= AX_UnitID[5], 
		tTimeout:= ParamTimeout,
		nQuantity		:= AX_QTY_MB[5] , 
		nMBAddr			:= AX_ADR_MB[5] ,  
		cbLength		:= SIZEOF(MesBlock5_Temp) , 
		pDestAddr		:= ADR(MesBlock5_Temp) , 
		ModbusReadAlarm	=>AX_ModbusReadAlarm[5] , 
		ErrorId			=> AX_ModbusReadAlarmId[5]
	);
	
	FB_ModbusRead[6]
	(
		nTCPPort	:= ParamTcpPort,
		ClockRead:= MesDataExd.MesData.MesCP_Read AND ClockRead, 
		Reset:= CmdClearFault_G OR IN_CmdReset_L,
		sIPAddr:=ParamIPAddress , 
		nUnitID:= AX_UnitID[6], 
		tTimeout:= ParamTimeout,
		nQuantity		:= AX_QTY_MB[6] , 
		nMBAddr			:= AX_ADR_MB[6] , 
		cbLength		:= SIZEOF(MesBlock6_Temp)  , 
		pDestAddr		:= ADR(MesBlock6_Temp) , 
		ModbusReadAlarm	=> AX_ModbusReadAlarm[6] , 
		ErrorId			=> AX_ModbusReadAlarmId[6]
	);
	
	*)
	// LOOP over all SSM Sunny String Monitor
	
		FB_ModbusRead[7]
	(
		nTCPPort	:= ParamTcpPort,
		ClockRead:= MesDataExd.MesData.MesCP_Read AND ClockRead ,  
		Reset:= CmdClearFault_G OR IN_CmdReset_L,
		sIPAddr:=ParamIPAddress , 
		nUnitID:= ParamUnitID_SSM[ID_SSM ] , 
		tTimeout:= ParamTimeout,
		nQuantity		:= AX_QTY_MB[7] , 
		nMBAddr			:= AX_ADR_MB[7] , 
		cbLength		:= SIZEOF(MesBlock7_Temp)  , 
		pDestAddr		:= ADR(MesBlock7_Temp) , 
		ModbusReadAlarm	=> AX_ModbusReadAlarm[7] , 
		ErrorId			=> AX_ModbusReadAlarmId[7]
	);
	

	
	
	
//			FB_ModbusRead[8]
//	(
//		nTCPPort	:= ParamTcpPort,
//		ClockRead:= MesDataExd.MesData.MesCP_Read AND ClockRead, 
//		Reset:= CmdClearFault_G OR IN_CmdReset_L,
//		sIPAddr:=ParamIPAddress , 
//		nUnitID:= AX_UnitID[8], 
//		tTimeout:= ParamTimeout,
//		nQuantity		:= AX_QTY_MB[8] , 
//		nMBAddr			:= AX_ADR_MB[8] , 
//		cbLength		:= SIZEOF(MesBlock8_Temp)  , 
//		pDestAddr		:= ADR(MesBlock8_Temp) , 
//		ModbusReadAlarm	=> AX_ModbusReadAlarm[8] , 
//		ErrorId			=> AX_ModbusReadAlarmId[8]
//	);
	

	
	
	MW(WORD_STRONG :=  MesBlock1_Temp[2  ],	WORD_WEAK := MesBlock1_Temp[1  ], SIZE := 2, FIX := 0, SIGNED := 0, VAR_OUT	:= MesDataExd.MesEventID);
	MW(WORD_STRONG :=  MesBlock1_Temp[4  ],	WORD_WEAK := MesBlock1_Temp[3  ], SIZE := 2, FIX := 0, SIGNED := 0, VAR_OUT	:= TimeInterm);	   
	MesDataExd.MesWaitGridTm := REAL_TO_TIME(TimeInterm*1000);
	MW(WORD_STRONG :=  MesBlock1_Temp[15 ],	WORD_WEAK := MesBlock1_Temp[16 ], SIZE := 2, FIX := 0, SIGNED := 0, VAR_OUT	:= MesDataExd.SetptRecoAction);	
	MW(WORD_STRONG :=  MesBlock1_Temp[21 ],	WORD_WEAK := MesBlock1_Temp[22 ], SIZE := 2, FIX := 0, SIGNED := 0, VAR_OUT	:= PosInterm);	
	MesDataExd.MesOpened_CBGrid := SEL(PosInterm=51,SEL(PosInterm=311,FALSE, TRUE), FALSE);
	MW(WORD_STRONG :=  MesBlock1_Temp[29 ],	WORD_WEAK := MesBlock1_Temp[30 ], SIZE := 2, FIX := 3, SIGNED := 0, VAR_OUT	:= MesDataExd.MesData.MesInsuResistor);
	MW(WORD_STRONG :=  MesBlock1_Temp[30 ],	WORD_WEAK := MesBlock1_Temp[31 ], SIZE := 2, FIX := 0, SIGNED := 0, VAR_OUT	:= PosInterm);	
	MesDataExd.MesState_KeyComut := SEL(PosInterm=381,SEL(PosInterm=569,FALSE, TRUE), FALSE);
	MW(WORD_STRONG :=  MesBlock1_Temp[45 ],	WORD_WEAK := MesBlock1_Temp[46 ], SIZE := 2, FIX := 0, SIGNED := 0, VAR_OUT	:= MesDataExd.MesState_Inv);	
	MW(WORD_STRONG :=  MesBlock1_Temp[47 ],	WORD_WEAK := MesBlock1_Temp[58 ], SIZE := 2, FIX := 0, SIGNED := 0, VAR_OUT	:= MesDataExd.MesIDError);	
	MW(WORD_STRONG :=  MesBlock1_Temp[51 ],	WORD_WEAK := MesBlock1_Temp[52 ], SIZE := 2, FIX := 0, SIGNED := 0, VAR_OUT	:= MesDataExd.MesEventID_INVSMA);	
	MW(WORD_STRONG :=  MesBlock1_Temp[53 ],	WORD_WEAK := MesBlock1_Temp[54 ], SIZE := 2, FIX := 0, SIGNED := 0, VAR_OUT	:= PosInterm);	
	MesDataExd.MesOpened_GFDI := SEL(PosInterm=51,SEL(PosInterm=311,FALSE, TRUE), FALSE);
	MW(WORD_STRONG :=  MesBlock1_Temp[55 ],	WORD_WEAK := MesBlock1_Temp[56 ], SIZE := 2, FIX := 0, SIGNED := 0, VAR_OUT	:= MesDataExd.MesState_Restart);	
	MW(WORD_STRONG :=  MesBlock1_Temp[61 ],	WORD_WEAK := MesBlock1_Temp[62 ], SIZE := 2, FIX := 0, SIGNED := 0, VAR_OUT	:= PosInterm);	
	MesDataExd.Mesdata.MesOpened_Dc := SEL(PosInterm=51,SEL(PosInterm=311,FALSE, TRUE), FALSE);
	MW(WORD_STRONG :=  MesBlock1_Temp[69 ],	WORD_WEAK := MesBlock1_Temp[70 ], SIZE := 2, FIX := 0, SIGNED := 0, VAR_OUT	:= PosInterm);	
	MesDataExd.Mesdata.MesOpened_Ac := SEL(PosInterm=51,SEL(PosInterm=311,FALSE, TRUE), FALSE);

	

	MW(WORD_STRONG :=  MesBlock2_Temp[2  ],	WORD_WEAK := MesBlock2_Temp[1  ], SIZE := 2, FIX := 0, SIGNED := 0, VAR_OUT	:= MesDataExd.MesEActTot);
	MW(WORD_STRONG :=  MesBlock2_Temp[4  ],	WORD_WEAK := MesBlock2_Temp[3  ], SIZE := 2, FIX := 0, SIGNED := 0, VAR_OUT	:= MesDataExd.MesEActDay);
	MW(WORD_STRONG :=  MesBlock2_Temp[29 ],	WORD_WEAK := MesBlock2_Temp[30 ], SIZE := 2, FIX := 0, SIGNED := 0, VAR_OUT	:= TimeInterm);
	MesDataExd.MesWorkingHr := REAL_TO_TIME(TimeInterm*1000);
	MW(WORD_STRONG :=  MesBlock2_Temp[31 ],	WORD_WEAK := MesBlock2_Temp[32 ], SIZE := 2, FIX := 0, SIGNED := 0, VAR_OUT	:= TimeInterm);
	MesDataExd.MesFeedTm := REAL_TO_TIME(TimeInterm*1000);
	MW(WORD_STRONG :=  MesBlock2_Temp[33 ],	WORD_WEAK := MesBlock2_Temp[34 ], SIZE := 2, FIX := 0, SIGNED := 0, VAR_OUT	:= TimeInterm);
	MesDataExd.MesWorkingHr_Fan1 := REAL_TO_TIME(TimeInterm*1000);
	MW(WORD_STRONG :=  MesBlock2_Temp[35 ],	WORD_WEAK := MesBlock2_Temp[36 ], SIZE := 2, FIX := 0, SIGNED := 0, VAR_OUT	:= TimeInterm);
	MesDataExd.MesWorkingHr_Fan2 := REAL_TO_TIME(TimeInterm*1000);
	MW(WORD_STRONG :=  MesBlock2_Temp[37 ],	WORD_WEAK := MesBlock2_Temp[38 ], SIZE := 2, FIX := 0, SIGNED := 0, VAR_OUT	:= TimeInterm);
	MesDataExd.MesWorkingHr_Fan3 := REAL_TO_TIME(TimeInterm*1000);
	MW(WORD_STRONG :=  MesBlock2_Temp[39 ],	WORD_WEAK := MesBlock2_Temp[40 ], SIZE := 2, FIX := 0, SIGNED := 0, VAR_OUT	:= TimeInterm);
	MesDataExd.MesWorkingHr_Heat := REAL_TO_TIME(TimeInterm*1000);
	MW(WORD_STRONG :=  MesBlock2_Temp[45 ],	WORD_WEAK := MesBlock2_Temp[46 ], SIZE := 2, FIX := 0, SIGNED := 0, VAR_OUT	:= TimeInterm);
	MesDataExd.MesWorkingHr_Heat2 := REAL_TO_TIME(TimeInterm*1000);
	(*MW(WORD_STRONG :=  MesBlock2_Temp[89 ],	WORD_WEAK := MesBlock2_Temp[90 ], SIZE := 2, FIX := 0, SIGNED := 0, VAR_OUT	:= TimeInterm);
	MesDataExd.MesData.MesWorkingHrtFan3 := REAL_TO_TIME(TimeInterm*1000); *)
	

